C02769=2104.969600,339.035500,-753.612600,90.034588,0.916732,0.000000
C02770=2082.812600,339.026400,-753.612600,88.974616,0.372423,-0.005730
C02771=2027.650200,339.018600,-753.612600,90.756515,-0.183346,-0.000000
C02772=1998.073600,339.007800,-753.612600,89.897078,-0.343775,0.000000
C02773=2074.825300,338.992600,-753.612600,89.358498,1.186023,-0.011459
C02774=2089.149900,338.987500,-753.612600,90.051777,-0.590147,-0.000000
C02775=2053.323900,338.978400,-753.612600,90.332526,-0.332316,-0.000000
C02776=2097.125300,338.974400,-753.612600,90.704949,-0.578687,-0.005730
C02777=2022.267800,338.959500,-753.612600,90.315337,-0.269290,-0.000000
C02778=2024.850700,338.932800,-753.612600,91.318013,0.355234,0.005730
C02779=2085.333300,338.914900,-753.612600,89.891348,0.166158,-0.000000
C02780=2038.206800,338.906800,-753.612600,89.971563,-0.320856,0.000000
C02781=2066.504500,338.886900,-753.612600,90.120532,-0.005730,-0.000000
C02782=2093.534600,338.865200,-753.612600,89.822594,0.091673,-0.000000
C02783=2058.436200,338.801600,-753.612600,90.131991,-0.676090,-0.000000
C02784=2073.063100,338.735200,-803.612600,90.343985,-0.807870,-0.005730
C02785=2062.264800,338.781500,-803.612600,89.364227,0.481285,-0.005730
C02786=2061.218800,338.791200,-803.612600,89.547574,-0.211994,0.000000
C02787=1999.241300,338.815900,-803.612600,88.779810,1.260507,-0.028648
C02788=2061.161000,338.858500,-803.612600,89.203799,0.275020,-0.005730
C02789=2096.996700,338.867600,-803.612600,88.808458,0.372423,-0.005730
C02790=2032.901900,338.882800,-803.612600,89.942915,-0.309397,0.000000
C02791=2104.217500,338.888900,-803.612600,91.174774,1.598552,0.034377
C02792=2019.781000,338.898300,-803.612600,89.587681,0.275020,-0.000000
C02793=2032.219500,338.910500,-803.612600,89.564763,-0.017189,0.000000
C02794=2088.973100,338.917600,-803.612600,90.195016,0.051566,0.000000
C02795=2038.272700,338.924400,-803.612600,89.834053,-0.177617,0.000000
C02796=2014.609200,338.933100,-803.612600,89.862701,-0.252101,0.000000
C02797=2100.091200,338.939200,-803.612600,90.974239,-0.315127,-0.005730
C02798=2046.154000,338.945000,-803.612600,90.842458,-0.807870,-0.011459
C02799=2077.330300,338.949000,-803.612600,89.856971,-0.286479,0.000000
C02800=2071.967600,338.953400,-803.612600,89.742379,0.160428,-0.000000
C02801=1988.870200,338.964600,-803.612600,90.114802,-0.504203,-0.000000
C02802=2111.765200,338.974700,-803.612600,89.983022,0.601606,-0.000000
C02803=2118.654200,338.987200,-803.612600,89.828323,0.068755,-0.000000
C02804=2105.787000,338.990900,-803.612600,90.407010,0.309397,0.000000
C02805=2049.676000,338.996000,-803.612600,90.235123,-0.487014,-0.000000
C02806=2122.801600,339.002700,-803.612600,90.143450,0.521392,0.000000
C02807=1998.518300,339.016900,-803.612600,89.977292,-0.137510,0.000000
C02808=2159.190800,339.028100,-803.612600,90.349715,0.446907,0.000000
C02809=2102.381000,339.034800,-803.612600,90.366903,0.452637,0.005730
C02810=2042.336700,339.040600,-803.612600,89.874160,0.429718,-0.000000
C02811=2113.548000,339.047700,-803.612600,90.143450,0.051566,0.000000
C02812=2131.010900,339.059800,-803.612600,89.484548,0.452637,-0.005730
C02813=1990.465400,339.066600,-803.612600,90.670571,-0.521392,-0.005730
C02814=2154.185700,339.079400,-803.612600,90.492954,0.257831,0.000000
C02815=2103.755700,339.090200,-803.612600,89.879889,0.349504,-0.000000
C02816=1978.876200,339.102600,-803.612600,89.604870,-0.160428,0.000000
C02817=2108.690000,339.109500,-803.612600,89.736650,0.521392,-0.000000
C02818=2117.282000,339.118300,-803.612600,89.157963,0.985487,-0.017189
C02819=2167.864000,339.126700,-803.612600,90.470036,0.469825,0.005730
C02820=1968.699400,339.144300,-803.612600,89.937185,-0.521392,0.000000
C02821=1980.830900,339.149400,-803.612600,89.553303,-0.635983,0.005730
C02822=2012.761200,339.158500,-803.612600,89.312661,-0.234913,0.000000
C02823=1979.519700,339.173400,-803.612600,89.215258,-0.395341,0.005730
C02824=2133.101400,339.181100,-803.612600,90.068965,-0.487014,-0.000000
C02825=2139.307800,339.203900,-803.612600,90.200746,0.721927,0.000000
C02826=2189.894000,339.212200,-803.612600,90.865377,-6.107730,-0.091673
C02827=2164.407500,339.218300,-803.612600,90.779433,-0.131780,-0.000000
C02828=1973.765200,339.226700,-803.612600,88.997534,0.051566,-0.000000
C02829=1963.063900,339.232100,-803.612600,89.793946,-0.120321,0.000000
C02830=2140.823500,339.248700,-803.612600,89.284013,0.693279,-0.011459
C02831=1966.561300,339.257100,-803.612600,90.441388,-0.721927,-0.005730
C02832=2146.546600,339.275400,-803.612600,89.736650,0.469825,-0.000000
C02833=1944.493700,339.305100,-803.612600,89.650706,-0.395341,0.000000
C02834=2164.597400,339.332800,-803.612600,90.934132,0.681820,0.011459
C02835=2179.742100,339.345000,-803.612600,90.630464,1.953786,0.022918
C02836=1959.256700,339.353400,-803.612600,89.845512,-0.315127,0.000000
C02837=1951.206300,339.375000,-803.612600,90.252312,-0.635983,-0.000000
C02838=1940.398000,339.403100,-803.612600,89.839782,-0.590147,0.000000
C02839=1952.858800,339.430500,-803.612600,90.269501,-0.103132,-0.000000
C02840=1940.391000,339.450700,-803.612600,90.172098,-0.676090,-0.000000
C02841=1925.004100,339.506500,-803.612600,90.000210,-0.441178,-0.000000
C02842=1931.783000,339.527400,-803.612600,89.839782,-0.257831,0.000000
C02843=1915.754700,339.565900,-803.612600,89.914267,-0.292208,0.000000
C02844=1925.891500,339.622000,-803.612600,89.541844,-0.538580,0.005730
C02845=1939.013200,339.694600,-803.612600,89.897078,-0.034377,0.000000
C02846=1916.706300,339.756800,-803.612600,90.017399,-0.847978,-0.000000
C02847=1906.137300,339.800400,-803.612600,89.685084,-0.762034,0.005730
C02848=1908.335200,339.879800,-803.612600,89.455901,-0.498473,0.005730
C02849=1891.927500,339.960500,-803.612600,89.748109,-0.985487,0.005730
C02850=1898.280800,340.042000,-803.612600,89.553303,-0.985487,0.005730
C02851=1878.249000,340.138700,-803.612600,90.017399,-1.254778,-0.000000
C02852=1890.381300,340.206100,-803.612600,90.601816,0.406800,0.005730
C02853=1874.073900,340.238200,-803.612600,89.759568,-1.203211,0.005730
C02854=1872.070100,340.338200,-803.612600,89.742379,-0.527121,0.000000
C02855=1878.439100,340.425700,-803.612600,89.983022,-0.842248,0.000000
C02856=1863.563200,340.545000,-803.612600,89.811134,-1.157375,0.005730
C02857=1858.204600,340.602100,-803.612600,90.051777,-1.037054,-0.000000
C02858=1846.137000,340.776800,-803.612600,89.375686,-1.048513,0.011459
C02859=1846.450600,340.848700,-803.612600,89.977292,-1.008406,0.000000
C02860=1839.612500,340.979500,-803.612600,89.146503,-0.355234,0.005730
C02861=1829.812800,341.022700,-803.612600,89.868430,-0.859437,0.000000
C02862=1794.925200,341.065000,-803.612600,91.100289,14.610424,0.280749
C02863=1837.928000,341.117300,-803.612600,89.467360,-0.658901,0.005730
C02864=1824.256700,341.181200,-803.612600,89.564763,-0.676090,0.005730
C02865=1817.402900,341.262300,-803.612600,89.450171,-1.312073,0.011459
C02866=1817.372500,341.325800,-803.612600,90.166368,-1.134456,-0.005730
C02867=1808.346600,341.423100,-803.612600,89.822594,-1.271966,0.005730
C02868=1812.505400,341.463600,-803.612600,89.576222,-1.180293,0.011459
C02869=1798.014800,341.534900,-803.612600,90.217934,5.460288,0.022918
C02870=1798.394100,341.571200,-803.612600,90.452847,4.497719,0.034377
C02871=1798.782000,341.649400,-803.612600,90.733596,3.254400,0.040107
C02872=1798.679300,341.821700,-853.612600,89.089208,2.366316,-0.040107
C02873=1801.796400,341.691700,-853.612600,90.384092,-0.332316,-0.000000
C02874=1803.834000,341.604200,-853.612600,91.358120,-1.976704,-0.045837
C02875=1797.252700,341.515600,-853.612600,93.718707,6.835386,0.441178
C02876=1811.298800,341.443300,-853.612600,90.481495,-1.999623,-0.017189
C02877=1813.044500,341.369400,-853.612600,90.074695,-1.930868,-0.000000
C02878=1814.433300,341.317300,-853.612600,90.510143,-1.673037,-0.017189
C02879=1816.535000,341.199100,-853.612600,90.057506,-0.893814,-0.000000
C02880=1822.945800,341.133500,-853.612600,89.685084,-1.220400,0.005730
C02881=1817.392400,341.111900,-853.612600,90.401281,-1.077161,-0.005730
C02882=1843.858500,340.985200,-853.612600,89.839782,-1.237589,0.005730
C02883=1842.018200,340.879500,-853.612600,90.412740,-1.249048,-0.011459
C02884=1843.463300,340.784900,-853.612600,90.017399,-0.435448,-0.000000
C02885=1850.351600,340.762600,-853.612600,89.954374,-0.888085,0.000000
C02886=1858.825800,340.665300,-853.612600,89.811134,-1.157375,0.005730
C02887=1864.859100,340.596000,-853.612600,89.135044,-0.011459,0.000000
C02888=1864.700800,340.570000,-853.612600,90.292419,-0.796411,-0.005730
C02889=1884.815000,340.449400,-853.612600,89.593410,-0.435448,0.005730
C02890=1866.700100,340.415900,-853.612600,90.945591,-0.733386,-0.011459
C02891=1875.256200,340.323000,-853.612600,90.292419,-0.481285,-0.000000
C02892=1889.321400,340.299700,-853.612600,89.576222,-0.739116,0.005730
C02893=1891.341900,340.243000,-853.612600,89.908537,-1.071431,0.000000
C02894=1897.280800,340.165900,-853.612600,90.848188,-0.635983,-0.011459
C02895=1904.713200,340.119000,-853.612600,89.215258,-0.378152,0.005730
C02896=1934.186200,340.090300,-853.612600,89.404334,-1.094349,0.011459
C02897=1904.887100,340.006800,-853.612600,89.444441,-0.572958,0.005730
C02898=1913.416700,339.981100,-853.612600,89.753839,-0.103132,0.000000
C02899=1924.127800,339.912600,-853.612600,90.607546,-0.045837,-0.000000
C02900=1952.628800,339.828100,-853.612600,87.404712,-0.063025,0.000000
C02901=1953.652400,339.784500,-853.612600,89.650706,-0.389611,0.000000
C02902=1947.297400,339.762600,-853.612600,89.587681,0.063025,-0.000000
C02903=1930.044800,339.732800,-853.612600,89.352768,-0.532851,0.005730
C02904=1937.784000,339.671000,-853.612600,88.819917,-1.014135,0.022918
C02905=1938.403200,339.637200,-853.612600,89.988751,-0.475555,0.000000
C02906=2047.261300,339.589900,-853.612600,77.377950,0.767763,-0.171887
C02907=1962.940900,339.523000,-853.612600,90.023129,-1.008406,-0.000000
C02908=1985.149800,339.488600,-853.612600,88.378740,-0.418259,0.011459
C02909=1981.144300,339.449700,-853.612600,90.023129,-0.613065,-0.000000
C02910=1957.762100,339.410500,-853.612600,89.679354,-0.378152,0.000000
C02911=1990.508900,339.405100,-853.612600,90.131991,-0.171887,-0.000000
C02912=2000.751600,339.354400,-853.612600,89.306932,-0.229183,0.000000
C02913=1982.854200,339.317900,-853.612600,88.739703,-0.492744,0.011459
C02914=2009.978300,339.297300,-853.612600,89.541844,0.767763,-0.005730
C02915=2024.539800,339.284800,-853.612600,90.051777,-0.257831,-0.000000
C02916=2121.511300,339.274700,-853.612600,88.407388,-0.303668,0.005730
C02917=2055.332600,339.230100,-853.612600,90.172098,0.532851,0.000000
C02918=2038.502000,339.213900,-853.612600,89.753839,-0.252101,0.000000
C02919=2083.289400,339.197800,-853.612600,89.352768,0.085944,-0.000000
C02920=1989.215900,339.185900,-853.612600,89.060560,-0.395341,0.005730
C02921=2067.307600,339.179100,-853.612600,89.908537,-0.842248,0.000000
C02922=2188.011000,339.171700,-853.612600,90.624734,-5.036299,-0.057296
C02923=2006.290800,339.150400,-853.612600,88.854295,0.303668,-0.005730
C02924=2087.059600,339.135500,-853.612600,90.939861,-0.842248,-0.011459
C02925=2182.180800,339.129800,-853.612600,89.753839,0.653172,-0.000000
C02926=2165.223600,339.123000,-853.612600,89.736650,0.739116,-0.005730
C02927=2179.411300,339.116900,-853.612600,74.570457,-0.538580,0.148969
C02928=2178.774900,339.105100,-853.612600,91.329473,-0.022918,-0.000000
C02929=1995.124200,339.097000,-853.612600,89.358498,-0.968299,0.011459
C02930=1998.114900,339.089200,-853.612600,90.796622,-0.853707,-0.011459
C02931=2028.129200,339.081800,-853.612600,91.615951,0.332316,0.011459
C02932=2071.745200,339.075700,-853.612600,89.610599,-0.607335,0.005730
C02933=2107.939900,339.069000,-853.612600,90.160639,0.183346,0.000000
C02934=2171.816500,339.059200,-853.612600,89.644977,-0.481285,0.005730
C02935=2006.319000,339.054400,-853.612600,90.716408,-0.441178,-0.005730
C02936=2061.621400,339.046000,-853.612600,89.937185,-0.097403,0.000000
C02937=2092.362100,339.039600,-853.612600,89.650706,-0.687549,0.005730
C02938=2127.230200,339.028800,-853.612600,90.653382,-0.297938,-0.005730
C02939=2142.220100,339.022000,-853.612600,90.080425,0.131780,0.000000
C02940=2050.404100,339.012200,-853.612600,90.366903,-0.097403,-0.000000
C02941=2017.120700,339.008500,-853.612600,91.008616,-0.148969,-0.000000
C02942=2097.055900,339.005400,-853.612600,90.745056,-1.082890,-0.011459
C02943=2146.699300,338.996700,-853.612600,90.195016,-0.378152,-0.000000
C02944=2169.661400,338.991300,-853.612600,90.212205,-0.509932,-0.000000
C02945=2155.902900,338.977700,-853.612600,90.372633,-0.211994,-0.000000
C02946=2135.683800,338.961200,-853.612600,89.862701,0.143239,-0.000000
C02947=2045.946900,338.948700,-853.612600,88.779810,0.819330,-0.017189
C02948=2091.307700,338.939600,-853.612600,89.392875,-0.252101,0.000000
C02949=2072.474700,338.934500,-853.612600,89.994481,-0.956840,0.000000
C02950=2109.023200,338.915600,-853.612600,89.496008,-0.223454,0.000000
C02951=2059.240800,338.906500,-853.612600,89.421523,-0.676090,0.005730
C02952=2189.032800,338.897000,-853.612600,92.091506,-4.251347,-0.154699
C02953=2113.653700,338.883800,-853.612600,90.825270,0.189076,0.000000
C02954=2114.931100,338.865200,-853.612600,85.806159,-0.234913,0.017189
C02955=2141.954900,338.841900,-853.612600,87.324498,-0.137510,0.005730
C02956=2158.166400,338.775700,-853.612600,91.363850,-0.068755,-0.000000
C02957=2182.832600,338.676000,-853.612600,93.770273,-0.269290,-0.017189
C02958=2192.460800,338.381800,-853.612600,92.859270,-14.661990,-0.727656
C02959=1845.943900,-262.579400,-444.761500,-85.135799,-0.796411,179.931666
C02960=2103.620100,-262.360400,-444.761500,-77.847776,0.338045,-179.925936
C02961=2106.924000,-262.167000,-444.761500,-88.086531,0.275020,-179.988962
C02962=1869.037500,-262.039800,-444.761500,-79.022339,1.271966,-179.754049
C02963=2042.284100,-262.001000,-444.761500,-86.321821,1.495420,-179.903018
C02964=2099.976800,-261.979000,-444.761500,-88.579275,1.363640,-179.966043
C02965=2077.569800,-261.892900,-444.761500,-79.474976,-0.378152,179.931666
C02966=2056.224500,-261.862800,-444.761500,-82.248091,-0.555769,179.925936
C02967=1929.876800,-261.815500,-444.761500,-82.654892,1.392287,-179.822804
C02968=1953.938600,-261.752700,-444.761500,-78.403545,-0.784952,179.839993
C02969=2043.564000,-261.713100,-444.761500,-75.722102,-0.802141,179.794156
C02970=1974.190100,-261.625300,-444.761500,-78.667105,-1.673037,179.662376
C02971=1921.842500,-260.819200,-494.761500,-91.965456,0.177617,179.994691
C02972=1911.461000,-260.905300,-494.761500,-92.211828,-0.572958,-179.977503
C02973=1866.999900,-260.969200,-494.761500,-92.165991,-0.613065,-179.977503
C02974=1870.542800,-261.046200,-494.761500,-91.885242,-0.303668,-179.988962
C02975=1916.503500,-261.073900,-494.761500,-91.535737,0.429718,179.988962
C02976=1861.862700,-261.137800,-494.761500,-92.074318,-0.951110,-179.966043
C02977=1937.964400,-261.156000,-494.761500,-91.696166,0.189076,179.994691
C02978=1998.654800,-261.175600,-494.761500,-91.197692,0.206265,179.994691
C02979=2020.094000,-261.188100,-494.761500,-91.535737,-0.423989,-179.988962
C02980=1933.449000,-261.219500,-494.761500,-92.842081,0.154699,179.994691
C02981=2024.472000,-261.238800,-494.761500,-92.343608,-0.120321,-179.994691
C02982=2016.615400,-261.241800,-494.761500,-91.512819,0.263561,179.994691
C02983=1957.998500,-261.260400,-494.761500,-91.742002,0.487014,179.983232
C02984=2090.231400,-261.293500,-494.761500,-91.873782,-0.183346,-179.994691
C02985=1857.870400,-261.303700,-494.761500,-90.899754,0.252101,179.994691
C02986=1869.562400,-261.332000,-494.761500,-91.106019,0.160428,179.994691
C02987=1956.272500,-261.355000,-494.761500,-92.269123,-0.063025,-179.994691
C02988=1980.693200,-261.373900,-494.761500,-91.226340,-0.532851,-179.988962
C02989=2081.434100,-261.394200,-494.761500,-91.060182,-0.022918,-180.000421
C02990=1849.814100,-261.409700,-494.761500,-91.633140,-0.108862,-179.994691
C02991=1898.632500,-261.421900,-494.761500,-91.151856,-0.200535,-179.994691
C02992=2077.098900,-261.431000,-494.761500,-91.128937,-0.647442,-179.988962
C02993=2080.090000,-261.448600,-494.761500,-90.997157,-0.269290,-179.994691
C02994=1868.275200,-261.460100,-494.761500,-91.661788,-0.601606,-179.983232
C02995=1897.656500,-261.478300,-494.761500,-92.498306,2.171510,179.903018
C02996=2006.452600,-261.495900,-494.761500,-91.925349,0.005730,180.000421
C02997=2097.180900,-261.502000,-494.761500,-91.432605,0.275020,179.994691
C02998=2003.950400,-261.515800,-494.761500,-90.378363,0.418259,179.994691
C02999=1974.234800,-261.535800,-494.761500,-90.659112,-0.143239,-180.000421
C03000=2124.803700,-261.548600,-494.761500,-91.656058,0.303668,179.988962
C03001=2094.531400,-261.564500,-494.761500,-90.767974,0.544310,179.994691
C03002=2132.074300,-261.573300,-494.761500,-91.214881,0.338045,179.994691
C03003=1884.756500,-261.584700,-494.761500,-92.647275,-0.567228,-179.971773
C03004=1949.279300,-261.598900,-494.761500,-90.682030,0.498473,179.994691
C03005=1986.413600,-261.603300,-494.761500,-91.329473,0.945380,179.977503
C03006=2088.847000,-261.615200,-494.761500,-90.699219,-0.630254,-179.994691
C03007=1907.677900,-261.626000,-494.761500,-91.323743,-0.217724,-179.994691
C03008=2055.490900,-261.635100,-494.761500,-90.401281,-0.028648,-180.000421
C03009=2026.414700,-261.643900,-494.761500,-90.361174,-0.269290,-180.000421
C03010=2116.655000,-261.651600,-494.761500,-90.504413,0.750575,179.994691
C03011=1933.336100,-261.663800,-494.761500,-91.048723,0.137510,179.994691
C03012=2092.292200,-261.669400,-494.761500,-92.246205,-0.085944,-179.994691
C03013=1945.953800,-261.681700,-494.761500,-91.593033,0.303668,179.988962
C03014=2022.229100,-261.689400,-494.761500,-90.555980,0.492744,179.994691
C03015=2193.443100,-261.697900,-494.761500,-92.630087,-7.563043,-179.656646
C03016=1994.152200,-261.709100,-494.761500,-90.922673,-0.773493,-179.988962
C03017=2117.856500,-261.713800,-494.761500,-90.945591,0.882355,179.983232
C03018=2150.660200,-261.719500,-494.761500,-91.128937,0.126051,180.000421
C03019=2026.671700,-261.724300,-494.761500,-90.212205,0.676090,179.994691
C03020=2181.140100,-261.730400,-494.761500,-89.427253,0.578687,-179.994691
C03021=1954.378200,-261.737500,-494.761500,-90.882565,0.584417,179.988962
C03022=2027.263400,-261.740800,-494.761500,-91.873782,-0.154699,-179.994691
C03023=1902.290500,-261.748100,-494.761500,-91.203422,-0.080214,-180.000421
C03024=2083.758200,-261.758100,-494.761500,-90.332526,-0.498473,-179.994691
C03025=1968.561800,-261.766200,-494.761500,-89.295472,-0.406800,179.994691
C03026=2142.714000,-261.772900,-494.761500,-90.876836,0.452637,179.994691
C03027=2013.614300,-261.780700,-494.761500,-90.836729,-0.796411,-179.988962
C03028=2071.154100,-261.790200,-494.761500,-91.186233,0.275020,179.994691
C03029=2077.380200,-261.803300,-494.761500,-91.644599,0.561499,179.983232
C03030=1914.243800,-261.809100,-494.761500,-90.458577,-0.676090,-179.994691
C03031=2162.444100,-261.814100,-494.761500,-90.916943,0.240642,179.994691
C03032=1989.357100,-261.816500,-494.761500,-90.664842,1.077161,179.988962
C03033=1909.275700,-261.821600,-494.761500,-91.014346,0.074485,180.000421
C03034=2185.796500,-261.830800,-494.761500,-89.954374,0.051566,-180.000421
C03035=1910.961200,-261.834800,-494.761500,-91.415416,-0.103132,-179.994691
C03036=2170.544700,-261.840800,-494.761500,-89.238177,-0.200535,179.994691
C03037=2169.153300,-261.845900,-494.761500,-89.971563,-0.315127,180.000421
C03038=1865.804400,-261.849300,-494.761500,-92.097236,0.647442,179.977503
C03039=1816.495600,-261.851000,-494.761500,-91.850864,-0.899544,-179.971773
C03040=2024.305000,-261.859400,-494.761500,-91.111749,0.229183,179.994691
C03041=2124.318800,-261.865500,-494.761500,-90.934132,0.246372,179.994691
C03042=2080.300500,-261.872100,-494.761500,-90.464306,-0.355234,-179.994691
C03043=2042.447100,-261.881500,-494.761500,-90.229394,-0.326586,-180.000421
C03044=1805.058100,-261.884400,-494.761500,-92.097236,-1.604282,-179.943125
C03045=2172.081100,-261.890800,-494.761500,-90.555980,-0.051566,-180.000421
C03046=2035.399300,-261.894500,-494.761500,-91.071642,0.257831,179.994691
C03047=2175.348700,-261.898300,-494.761500,-90.825270,-0.320856,-179.994691
C03048=2190.438600,-261.904700,-494.761500,-88.986075,-0.951110,179.983232
C03049=2165.547600,-261.916800,-494.761500,-89.983022,-0.853707,180.000421
C03050=2188.317000,-261.922600,-494.761500,-90.452847,0.355234,179.994691
C03051=1810.669700,-261.930200,-494.761500,-91.707625,-1.346451,-179.960314
C03052=2095.544100,-261.934100,-494.761500,-90.762244,-0.870896,-179.988962
C03053=2113.841200,-261.939100,-494.761500,-88.819917,0.315127,-179.994691
C03054=2047.699800,-261.949300,-494.761500,-90.321067,-0.114592,-180.000421
C03055=2038.089400,-261.958100,-494.761500,-89.513196,-0.005730,180.000421
C03056=2022.620600,-261.962800,-494.761500,-90.704949,-0.292208,-179.994691
C03057=2141.279100,-261.973300,-494.761500,-90.177827,0.951110,179.994691
C03058=1879.830200,-261.982700,-494.761500,-91.346661,0.383882,179.988962
C03059=2077.005200,-262.004700,-494.761500,-90.361174,0.028648,180.000421
C03060=1821.697300,-262.022900,-494.761500,-91.180504,-0.687549,-179.983232
C03061=2102.265300,-262.033400,-494.761500,-90.091884,0.091673,180.000421
C03062=1839.440400,-262.042200,-494.761500,-91.638870,0.171887,179.994691
C03063=1920.936600,-262.050300,-494.761500,-84.408142,-0.974028,179.903018
C03064=1848.899200,-262.065200,-494.761500,-89.347039,-1.753251,179.977503
C03065=1811.781100,-262.089400,-494.761500,-91.157585,-1.048513,-179.977503
C03066=1805.613700,-262.106400,-494.761500,-90.767974,-1.283425,-179.983232
C03067=2144.861100,-262.140200,-494.761500,-89.702272,0.166158,-180.000421
C03068=1811.431300,-262.204400,-494.761500,-90.109072,-1.277696,-179.994691
C03069=1863.241200,-262.289800,-494.761500,-90.882565,-0.303668,-179.994691
C03070=1831.979100,-262.356000,-494.761500,-93.277529,0.504203,179.971773
C03071=1796.446100,-262.384400,-494.761500,-90.578898,5.826981,179.943125
C03072=1847.265200,-262.436800,-494.761500,-91.060182,-1.100079,-179.977503
C03073=1818.793200,-262.555400,-494.761500,-91.489901,-0.796411,-179.977503
C03074=1801.917400,-262.590200,-494.761500,-91.862323,-1.340721,-179.954584
C03075=1806.287400,-262.817200,-494.761500,-77.418057,-2.326209,179.479029
C03076=2193.404700,-262.778700,-544.761500,-88.166746,1.770440,-179.943125
C03077=2189.447400,-261.928300,-544.761500,-90.813811,4.360209,179.937396
C03078=2190.414600,-261.848900,-544.761500,-90.619005,0.418259,179.994691
C03079=2184.051200,-261.800300,-544.761500,-89.960103,-1.048513,180.000421
C03080=2181.482000,-261.731400,-544.761500,-90.693489,0.699009,179.988962
C03081=2167.358100,-261.706900,-544.761500,-90.699219,-0.120321,-180.000421
C03082=2171.713400,-261.665800,-544.761500,-90.762244,0.126051,180.000421
C03083=2156.638400,-261.640200,-544.761500,-91.002887,0.744845,179.988962
C03084=2139.836100,-261.607700,-544.761500,-91.289365,0.137510,179.994691
C03085=1812.547300,-261.579000,-544.761500,-91.237799,-1.741792,-179.960314
C03086=2171.946200,-261.543500,-544.761500,-90.859647,1.231859,179.983232
C03087=2154.229600,-261.503000,-544.761500,-91.077371,0.699009,179.988962
C03088=2173.622000,-261.451600,-544.761500,-91.318013,0.693279,179.983232
C03089=1814.094900,-261.418500,-544.761500,-90.716408,-1.082890,-179.988962
C03090=1805.093300,-261.396200,-544.761500,-91.065912,-1.398017,-179.971773
C03091=2168.330700,-261.378000,-544.761500,-90.985698,1.025594,179.983232
C03092=1836.531800,-261.352000,-544.761500,-91.713354,-0.624524,-179.983232
C03093=2178.750100,-261.297200,-544.761500,-90.498684,1.741792,179.983232
C03094=2100.472100,-261.271900,-544.761500,-91.512819,0.263561,179.994691
C03095=2129.860700,-261.209700,-544.761500,-92.206098,0.355234,179.988962
C03096=1809.421600,-261.193900,-544.761500,-90.492954,-0.933921,-179.994691
C03097=2164.807600,-261.175600,-544.761500,-90.309608,1.306344,179.994691
C03098=1821.197500,-261.137100,-544.761500,-90.739326,-0.916732,-179.988962
C03099=2064.002700,-261.115500,-544.761500,-91.495630,-0.085944,-180.000421
C03100=1837.038600,-261.079700,-544.761500,-91.289365,-0.796411,-179.983232
C03101=2144.955900,-261.059100,-544.761500,-91.587304,0.670361,179.983232
C03102=1816.312600,-261.036800,-544.761500,-90.573168,-0.681820,-179.994691
C03103=2007.052200,-261.008700,-544.761500,-91.232070,1.289155,179.971773
C03104=1815.077400,-260.995200,-544.761500,-91.106019,-1.254778,-179.977503
C03105=2020.728300,-260.981300,-544.761500,-91.684706,0.401070,179.988962
C03106=1935.614200,-260.958400,-544.761500,-91.827946,0.395341,179.988962
C03107=1815.197000,-260.941800,-544.761500,-89.581951,-1.988164,179.983232
C03108=2038.539300,-260.917200,-544.761500,-92.377985,0.584417,179.977503
C03109=1995.584900,-260.905300,-544.761500,-92.693112,0.315127,179.983232
C03110=1821.920700,-260.891500,-544.761500,-91.111749,-1.157375,-179.977503
C03111=1972.452200,-260.872900,-544.761500,-91.661788,0.183346,179.994691
C03112=1871.622600,-260.855000,-544.761500,-91.839405,-0.223454,-179.994691
C03113=1992.617400,-260.839600,-544.761500,-93.162937,0.074485,179.994691
C03114=2131.634500,-260.824600,-544.761500,-91.656058,0.779223,179.977503
C03115=2035.438300,-260.806300,-544.761500,-91.037264,-0.933921,-179.983232
C03116=2114.512500,-260.763800,-544.761500,-91.421146,1.128727,179.971773
C03117=2078.864700,-260.750300,-544.761500,-92.171721,0.297938,179.988962
C03118=2157.676000,-260.733700,-544.761500,-91.318013,1.707414,179.960314
C03119=1866.480200,-260.724600,-544.761500,-91.226340,-0.647442,-179.988962
C03120=1988.083400,-260.707700,-544.761500,-91.805028,0.246372,179.994691
C03121=1978.238600,-260.688100,-544.761500,-91.673247,0.739116,179.977503
C03122=1897.058900,-260.662000,-544.761500,-92.859270,-1.306344,-179.937396
C03123=1825.113400,-260.652600,-544.761500,-90.876836,-0.951110,-179.983232
C03124=2095.767400,-260.644900,-544.761500,-91.633140,0.544310,179.983232
C03125=1876.881500,-260.633000,-544.761500,-92.836352,0.739116,179.966043
C03126=2074.786700,-260.610100,-544.761500,-92.194639,0.561499,179.977503
C03127=1924.829500,-260.589100,-544.761500,-91.186233,-0.389611,-179.994691
C03128=2116.875600,-260.582700,-544.761500,-91.976915,0.143239,179.994691
C03129=1842.483900,-260.561400,-544.761500,-91.163315,-1.243318,-179.977503
C03130=2027.544200,-260.536400,-544.761500,-91.873782,0.343775,179.988962
C03131=1850.823900,-260.517500,-544.761500,-91.243529,-0.068755,-180.000421
C03132=1875.209900,-260.495900,-544.761500,-91.902430,-0.177617,-179.994691
C03133=1971.870300,-260.470500,-544.761500,-91.363850,0.338045,179.994691
C03134=1987.957000,-260.444900,-544.761500,-91.174774,2.234535,179.954584
C03135=1835.514400,-260.423200,-544.761500,-89.919996,-0.968299,180.000421
C03136=1980.580000,-260.409000,-544.761500,-92.504036,-0.739116,-179.966043
C03137=1848.362100,-260.392500,-544.761500,-91.484171,-0.802141,-179.977503
C03138=1831.829900,-260.365800,-544.761500,-89.730920,-2.881978,179.988962
C03139=2135.648000,-260.354300,-544.761500,-91.403957,0.584417,179.983232
C03140=1920.149600,-260.334400,-544.761500,-92.137343,0.252101,179.988962
C03141=1873.512100,-260.317800,-544.761500,-91.083101,-0.515662,-179.988962
C03142=2090.011200,-260.305000,-544.761500,-92.097236,0.257831,179.988962
C03143=1999.619000,-260.288600,-544.761500,-91.501360,-0.097403,-179.994691
C03144=2118.771400,-260.267500,-544.761500,-91.232070,0.790682,179.983232
C03145=1893.437100,-260.253300,-544.761500,-91.598763,-0.303668,-179.988962
C03146=1995.325000,-260.237900,-544.761500,-92.635816,-0.206265,-179.988962
C03147=1877.827800,-260.217500,-544.761500,-91.363850,-1.111538,-179.971773
C03148=1861.590800,-260.198900,-544.761500,-92.114425,-0.561499,-179.977503
C03149=1949.022700,-260.188100,-544.761500,-91.931078,0.045837,180.000421
C03150=2065.874400,-260.160700,-544.761500,-92.188909,0.223454,179.988962
C03151=1984.529000,-260.117400,-544.761500,-91.638870,-0.418259,-179.988962
C03152=1946.014500,-260.067500,-544.761500,-91.919619,-0.085944,-179.994691
C03153=2028.490500,-260.046200,-544.761500,-90.945591,1.461042,179.977503
C03154=1878.387900,-260.014800,-544.761500,-91.495630,-1.134456,-179.971773
C03155=2054.593000,-260.005000,-544.761500,-92.750408,-0.332316,-179.983232
C03156=2072.406500,-259.984400,-544.761500,-92.429552,-0.022918,-180.000421
C03157=1954.819400,-259.971500,-544.761500,-92.767597,-0.349504,-179.983232
C03158=2079.669100,-259.920900,-544.761500,-92.148802,0.120321,179.994691
C03159=2034.819700,-259.900600,-544.761500,-92.830622,0.326586,179.983232
C03160=2001.013700,-259.884400,-544.761500,-90.727867,0.504203,179.994691
C03161=1936.039800,-259.870200,-544.761500,-92.412363,-0.389611,-179.983232
C03162=2016.505000,-259.830600,-544.761500,-91.461253,-1.329262,-179.966043
C03163=2105.713500,-259.797200,-544.761500,-92.292042,0.681820,179.971773
C03164=1928.160200,-259.790800,-544.761500,-92.337878,0.521392,179.977503
C03165=2100.667200,-259.760700,-544.761500,-92.589980,0.338045,179.983232
C03166=1968.585700,-259.715800,-544.761500,-92.549873,1.919409,179.914477
C03167=1957.890100,-259.692800,-544.761500,-92.446740,1.111538,179.954584
C03168=1907.944600,-259.650900,-544.761500,-92.412363,-0.928192,-179.960314
C03169=2022.531700,-259.635000,-544.761500,-91.644599,-0.269290,-179.994691
C03170=2045.046000,-259.595200,-544.761500,-91.879512,-0.882355,-179.971773
C03171=1945.854800,-259.558700,-544.761500,-93.816109,0.618794,179.960314
C03172=2035.480500,-259.537400,-544.761500,-92.229016,0.807870,179.966043
C03173=2051.644000,-259.510700,-544.761500,-92.504036,-0.784952,-179.966043
C03174=2087.205400,-259.470800,-544.761500,-91.232070,0.349504,179.994691
C03175=1976.162800,-259.450000,-544.761500,-93.374932,0.481285,179.971773
C03176=1946.439700,-259.404300,-544.761500,-91.673247,-0.114592,-179.994691
C03177=1957.313100,-259.374000,-544.761500,-92.028481,-0.498473,-179.983232
C03178=2083.156000,-259.348500,-544.761500,-90.762244,-0.040107,-180.000421
C03179=1979.022000,-259.233300,-544.761500,-90.722137,-0.120321,-180.000421
C03180=1975.506000,-257.856600,-594.761500,-92.108695,-0.389611,-179.983232
C03181=2006.601900,-257.960700,-594.761500,-91.552926,0.819330,179.977503
C03182=2043.583500,-257.974500,-594.761500,-90.796622,0.000000,180.000421
C03183=2076.505700,-257.997800,-594.761500,-91.191963,0.572958,179.988962
C03184=2005.853900,-258.029900,-594.761500,-91.999833,0.177617,179.994691
C03185=1968.632200,-258.047200,-594.761500,-91.020075,0.148969,179.994691
C03186=1950.789900,-258.061700,-594.761500,-91.650329,-0.171887,-179.994691
C03187=1936.259000,-258.086700,-594.761500,-91.117478,0.699009,179.988962
C03188=1945.613800,-258.125400,-594.761500,-91.959726,-1.804817,-179.937396
C03189=2075.447500,-258.155600,-594.761500,-91.123208,-0.080214,-180.000421
C03190=1950.546200,-258.173200,-594.761500,-92.383715,-0.664631,-179.971773
C03191=1926.315400,-258.193800,-594.761500,-90.767974,-0.383882,-179.994691
C03192=1982.653400,-258.200200,-594.761500,-90.596087,0.739116,179.994691
C03193=1978.382700,-258.235700,-594.761500,-91.959726,-0.103132,-179.994691
C03194=2019.060400,-258.261000,-594.761500,-91.547197,-0.103132,-179.994691
C03195=1947.702100,-258.288000,-594.761500,-91.295095,-0.034377,-180.000421
C03196=2010.528200,-258.308000,-594.761500,-90.636194,-0.590147,-179.994691
C03197=1974.208100,-258.315100,-594.761500,-91.386768,-0.246372,-179.994691
C03198=2047.057400,-258.336700,-594.761500,-90.756515,0.710468,179.988962
C03199=2110.855600,-258.380300,-594.761500,-90.533061,1.363640,179.988962
C03200=1897.268300,-258.412700,-594.761500,-91.077371,0.847978,179.983232
C03201=1934.923000,-258.446500,-594.761500,-90.928402,-0.211994,-179.994691
C03202=2062.708900,-258.475500,-594.761500,-92.876459,-1.008406,-179.948855
C03203=1991.921800,-258.489100,-594.761500,-90.991427,-0.040107,-180.000421
C03204=2071.862000,-258.515800,-594.761500,-91.438335,0.057296,180.000421
C03205=2077.376000,-258.534000,-594.761500,-92.068588,0.859437,179.971773
C03206=1885.348400,-258.538000,-594.761500,-89.702272,0.131780,-180.000421
C03207=1982.583000,-258.548200,-594.761500,-91.478442,-0.584417,-179.983232
C03208=1900.176200,-258.564700,-594.761500,-91.289365,-0.068755,-180.000421
C03209=1966.706900,-258.589400,-594.761500,-90.813811,0.762034,179.988962
C03210=2107.198600,-258.596500,-594.761500,-90.997157,0.458366,179.994691
C03211=2059.464300,-258.620500,-594.761500,-91.340932,-0.103132,-180.000421
C03212=1910.029600,-258.641800,-594.761500,-91.432605,-0.446907,-179.988962
C03213=2118.898600,-258.685700,-594.761500,-90.853918,1.289155,179.983232
C03214=1883.168600,-258.709000,-594.761500,-91.060182,-0.756304,-179.983232
C03215=2032.730800,-258.733300,-594.761500,-91.890971,0.338045,179.988962
C03216=2039.315900,-258.747200,-594.761500,-92.217557,0.011459,180.000421
C03217=1906.954400,-258.789700,-594.761500,-92.314960,0.189076,179.994691
C03218=2122.856000,-258.799900,-594.761500,-90.332526,1.569904,179.988962
C03219=1937.499100,-258.819800,-594.761500,-91.742002,0.429718,179.988962
C03220=2076.275000,-258.844800,-594.761500,-91.799298,0.607335,179.983232
C03221=2006.823400,-258.871500,-594.761500,-90.876836,0.223454,179.994691
C03222=1892.551100,-258.879900,-594.761500,-91.398227,-0.687549,-179.983232
C03223=2014.743300,-258.919500,-594.761500,-91.369580,0.584417,179.983232
C03224=2074.409200,-258.971800,-594.761500,-92.521225,0.355234,179.983232
C03225=1921.246800,-258.981000,-594.761500,-91.495630,0.045837,180.000421
C03226=2056.623300,-259.012400,-594.761500,-92.309230,0.790682,179.966043
C03227=1976.930800,-259.023200,-594.761500,-91.060182,-0.326586,-179.994691
C03228=1888.774200,-259.039100,-594.761500,-91.197692,-1.002676,-179.977503
C03229=1875.304000,-259.056300,-594.761500,-91.707625,-0.223454,-179.994691
C03230=1907.160300,-259.075600,-594.761500,-92.286312,0.017189,180.000421
C03231=1887.079600,-259.105600,-594.761500,-90.762244,-1.243318,-179.983232
C03232=1936.288600,-259.118800,-594.761500,-92.435281,0.383882,179.983232
C03233=2040.977100,-259.134300,-594.761500,-90.945591,-0.343775,-179.994691
C03234=2128.164300,-259.163700,-594.761500,-91.398227,1.300614,179.966043
C03235=2072.801000,-259.188400,-594.761500,-92.137343,0.429718,179.983232
C03236=1871.532200,-259.218100,-594.761500,-90.767974,-1.988164,-179.971773
C03237=2034.112800,-259.246800,-594.761500,-91.994104,-0.131780,-179.994691
C03238=1862.458300,-259.269800,-594.761500,-91.587304,-1.403747,-179.960314
C03239=1857.782200,-259.295500,-594.761500,-91.048723,-1.764710,-179.966043
C03240=1964.076700,-259.322500,-594.761500,-92.102966,0.767763,179.971773
C03241=2047.145300,-259.352600,-594.761500,-92.853540,-1.386558,-179.931666
C03242=1880.959500,-259.406300,-594.761500,-91.426875,-0.796411,-179.977503
C03243=2004.925400,-259.456300,-594.761500,-91.598763,0.928192,179.971773
C03244=2099.609400,-259.488400,-594.761500,-91.776380,2.051189,179.937396
C03245=2144.537300,-259.524200,-594.761500,-90.842458,2.354857,179.966043
C03246=2105.933800,-259.586700,-594.761500,-92.039940,0.595876,179.977503
C03247=1848.169700,-259.648900,-594.761500,-90.074695,-1.873572,-180.000421
C03248=1847.758100,-259.734400,-594.761500,-90.550250,-1.610011,-179.983232
C03249=2144.235100,-259.767100,-594.761500,-91.518549,2.515285,179.931666
C03250=1842.596100,-259.859400,-594.761500,-90.796622,-1.375099,-179.983232
C03251=2136.079200,-259.888100,-594.761500,-91.530008,1.575634,179.960314
C03252=2143.069900,-259.985700,-594.761500,-91.581574,1.541256,179.960314
C03253=1840.442500,-260.007300,-594.761500,-90.074695,-2.343397,-179.994691
C03254=1836.528600,-260.061400,-594.761500,-90.389822,-2.011082,-179.988962
C03255=2161.067000,-260.162800,-594.761500,-89.948644,3.277319,-179.994691
C03256=1833.421400,-260.234000,-594.761500,-90.349715,-2.761657,-179.983232
C03257=2156.691400,-260.301300,-594.761500,-91.318013,1.919409,179.954584
C03258=1828.131500,-260.435400,-594.761500,-90.487225,0.343775,179.994691
C03259=1822.949300,-260.521200,-594.761500,-90.401281,-2.320479,-179.983232
C03260=2169.354800,-260.567500,-594.761500,-90.000210,2.945003,180.000421
C03261=1820.066800,-260.698600,-594.761500,-89.771027,-1.873572,179.994691
C03262=1821.878900,-260.763800,-594.761500,-90.154909,-2.452259,-179.994691
C03263=1815.778300,-260.860400,-594.761500,-89.295472,-1.913679,179.977503
C03264=2176.814800,-260.934000,-594.761500,-90.676301,3.254400,179.960314
C03265=2172.570400,-260.978500,-594.761500,-90.567439,2.274642,179.977503
C03266=1809.014800,-261.035700,-594.761500,-90.005940,-2.062648,-180.000421
C03267=1812.378300,-261.091800,-594.761500,-89.994481,-2.486637,180.000421
C03268=1811.469600,-261.134100,-594.761500,-89.587681,-3.030947,179.977503
C03269=1806.242800,-261.193900,-594.761500,-89.129315,-2.354857,179.966043
C03270=1799.144000,-261.309100,-594.761500,-88.991805,-3.288778,179.943125
C03271=1796.063900,-261.353000,-594.761500,-88.126638,7.465640,-179.754049
C03272=1800.022000,-261.367200,-594.761500,-88.900131,-1.764710,179.966043
C03273=1802.737100,-261.531700,-594.761500,-89.381416,-3.065324,179.966043
C03274=1795.613900,-261.580000,-594.761500,-87.215636,0.653172,-179.966043
C03275=2187.688400,-261.652000,-594.761500,-89.856971,3.432017,-179.988962
C03276=1797.468200,-261.768900,-594.761500,-88.877213,-2.876248,179.943125
C03277=2190.839400,-261.875000,-594.761500,-91.031534,1.535527,179.971773
C03278=1797.016500,-261.995900,-594.761500,-88.860024,2.893437,-179.943125
C03279=1798.970800,-262.465800,-644.761500,-88.814188,-2.692902,179.943125
C03280=1796.247600,-262.211100,-644.761500,-89.547574,-0.401070,179.994691
C03281=2191.211700,-262.002300,-644.761500,-87.536492,-0.080214,179.994691
C03282=1803.707200,-261.891800,-644.761500,-89.679354,-5.993139,179.966043
C03283=1803.478200,-261.793900,-644.761500,-89.398605,-3.277319,179.966043
C03284=2187.072000,-261.722600,-644.761500,-88.825647,4.182592,-179.914477
C03285=2193.651900,-261.661800,-644.761500,-91.976915,-13.676503,-179.530596
C03286=2187.221700,-261.583900,-644.761500,-89.713732,3.460665,-179.983232
C03287=1804.257500,-261.440800,-644.761500,-90.544520,-4.572203,-179.954584
C03288=1811.483600,-261.369500,-644.761500,-89.077748,-3.982057,179.937396
C03289=1810.682200,-261.260800,-644.761500,-90.779433,-2.933544,-179.960314
C03290=2177.467100,-261.107200,-644.761500,-90.154909,3.827358,179.988962
C03291=2177.509300,-260.994500,-644.761500,-89.702272,3.179916,-179.983232
C03292=1821.215600,-260.865200,-644.761500,-90.097613,-2.927814,-179.994691
C03293=2172.041700,-260.749300,-644.761500,-89.742379,3.105431,-179.988962
C03294=2170.868000,-260.702800,-644.761500,-90.286689,3.093972,179.983232
C03295=1828.065600,-260.492800,-644.761500,-91.163315,-3.008028,-179.937396
C03296=1832.099000,-260.313800,-644.761500,-90.424199,-3.225752,-179.977503
C03297=2164.047100,-260.166500,-644.761500,-88.751162,2.796034,-179.937396
C03298=1836.783100,-260.034700,-644.761500,-89.627788,-2.589769,179.983232
C03299=2156.915300,-259.932300,-644.761500,-89.759568,2.635606,-179.988962
C03300=1842.827200,-259.797500,-644.761500,-90.149179,-3.168457,-179.988962
C03301=1836.341800,-259.756700,-644.761500,-91.323743,-1.776169,-179.960314
C03302=1845.845400,-259.557700,-644.761500,-89.392875,-3.970598,179.960314
C03303=1850.073800,-259.457700,-644.761500,-90.286689,-2.641335,-179.988962
C03304=1853.851300,-259.396200,-644.761500,-90.624734,-1.942327,-179.977503
C03305=1847.099300,-259.295200,-644.761500,-89.077748,-2.870519,179.954584
C03306=2141.896000,-259.242500,-644.761500,-89.673625,2.824682,-179.983232
C03307=1856.964600,-259.117800,-644.761500,-90.275230,-2.217347,-179.988962
C03308=1861.627400,-259.005600,-644.761500,-89.243906,-2.595499,179.966043
C03309=1859.827900,-258.931000,-644.761500,-90.510143,-2.171510,-179.983232
C03310=1871.831800,-258.822500,-644.761500,-90.057506,-1.764710,-180.000421
C03311=1865.678800,-258.764100,-644.761500,-89.427253,-1.598552,179.983232
C03312=2122.715500,-258.728600,-644.761500,-91.008616,1.363640,179.977503
C03313=2117.886100,-258.659000,-644.761500,-89.524655,2.034000,-179.983232
C03314=1871.010900,-258.626900,-644.761500,-90.292419,-2.383504,-179.988962
C03315=1876.193500,-258.563000,-644.761500,-91.421146,-1.718873,-179.954584
C03316=2116.714400,-258.509800,-644.761500,-91.209151,0.641713,179.988962
C03317=1885.146900,-258.430600,-644.761500,-91.988374,-1.885031,-179.937396
C03318=2114.671400,-258.362400,-644.761500,-90.189287,1.386558,179.994691
C03319=1872.610800,-258.298500,-644.761500,-90.848188,-1.701685,-179.977503
C03320=1882.136000,-258.248200,-644.761500,-89.559033,-1.822006,179.983232
C03321=1895.852800,-258.212700,-644.761500,-90.166368,-1.443854,-179.994691
C03322=1889.422500,-258.161400,-644.761500,-90.916943,-1.065701,-179.983232
C03323=2102.364000,-258.132500,-644.761500,-89.839782,0.773493,-180.000421
C03324=2101.942600,-258.108000,-644.761500,-90.126261,0.899544,180.000421
C03325=1899.936700,-258.068100,-644.761500,-90.407010,-1.082890,-179.994691
C03326=2103.695400,-258.025200,-644.761500,-89.788216,1.140186,-179.994691
C03327=2082.194000,-257.993100,-644.761500,-91.209151,1.443854,179.971773
C03328=2076.015400,-257.952900,-644.761500,-90.515872,0.727656,179.994691
C03329=1910.703300,-257.931300,-644.761500,-91.060182,-0.452637,-179.988962
C03330=1917.100900,-257.917700,-644.761500,-90.785163,-0.389611,-179.994691
C03331=1940.719100,-257.905200,-644.761500,-91.306554,-0.269290,-179.994691
C03332=1961.928100,-257.889700,-644.761500,-91.146126,0.263561,179.994691
C03333=2090.408800,-257.871800,-644.761500,-90.584627,0.939651,179.988962
C03334=2072.946000,-257.854600,-644.761500,-90.384092,1.340721,179.988962
C03335=1910.699500,-257.840400,-644.761500,-88.923050,0.905273,-179.983232
C03336=2023.164200,-257.823500,-644.761500,-91.002887,-0.017189,-180.000421
C03337=2084.155600,-257.804900,-644.761500,-90.813811,0.343775,179.994691
C03338=2012.223800,-257.788000,-644.761500,-91.593033,-0.034377,-180.000421
C03339=1936.512200,-257.780800,-644.761500,-90.670571,-0.223454,-179.994691
C03340=1919.876700,-257.759300,-644.761500,-90.750785,-0.853707,-179.988962
C03341=2002.111600,-257.748500,-644.761500,-90.246582,-0.664631,-179.994691
C03342=2018.400300,-257.732300,-644.761500,-91.123208,0.515662,179.988962
C03343=2064.837500,-257.722200,-644.761500,-89.793946,0.550039,-180.000421
C03344=2081.925200,-257.710300,-644.761500,-89.518926,0.366693,-179.994691
C03345=2037.211000,-257.700900,-644.761500,-90.429929,-0.916732,-179.994691
C03346=1993.727300,-257.689700,-644.761500,-91.426875,-0.103132,-179.994691
C03347=2001.922300,-257.685300,-644.761500,-90.997157,0.412530,179.994691
C03348=1930.788900,-257.678600,-644.761500,-91.289365,-0.521392,-179.988962
C03349=1900.989700,-257.669100,-644.761500,-91.449794,-0.796411,-179.977503
C03350=1937.710700,-257.660000,-644.761500,-90.682030,-0.418259,-179.994691
C03351=2083.356000,-257.652200,-644.761500,-90.252312,0.418259,180.000421
C03352=1967.410700,-257.646100,-644.761500,-91.169044,-0.297938,-179.994691
C03353=1925.347400,-257.641100,-644.761500,-90.538791,-0.825059,-179.994691
C03354=1958.648200,-257.624900,-644.761500,-91.008616,0.240642,179.994691
C03355=2037.434100,-257.617800,-644.761500,-91.254988,-0.080214,-180.000421
C03356=1899.387800,-257.605600,-644.761500,-90.504413,-1.346451,-179.988962
C03357=2025.422700,-257.589700,-644.761500,-92.011292,0.527121,179.983232
C03358=1975.027400,-257.575900,-644.761500,-91.913889,1.822006,179.937396
C03359=1915.038200,-257.549200,-644.761500,-90.349715,-0.676090,-179.994691
C03360=1972.643600,-257.539400,-644.761500,-91.031534,0.750575,179.988962
C03361=1959.202700,-257.523500,-644.761500,-91.031534,1.220400,179.977503
C03362=1951.110200,-257.510000,-644.761500,-90.212205,-0.011459,-180.000421
C03363=2010.252000,-257.502200,-644.761500,-89.392875,-0.515662,179.994691
C03364=1928.495500,-257.494400,-644.761500,-91.088830,0.378152,179.994691
C03365=2029.678300,-257.485000,-644.761500,-91.094560,-0.452637,-179.988962
C03366=1953.653200,-257.474800,-644.761500,-90.057506,-0.320856,-180.000421
C03367=1941.790800,-257.458300,-644.761500,-90.412740,-0.017189,-180.000421
C03368=2020.357300,-257.444100,-644.761500,-90.246582,0.389611,180.000421
C03369=2043.800600,-257.430600,-644.761500,-89.547574,-1.122997,179.988962
C03370=1953.336000,-257.408000,-644.761500,-91.037264,0.080214,180.000421
C03371=1974.292200,-257.387300,-644.761500,-89.965833,0.120321,-180.000421
C03372=1965.413900,-257.369800,-644.761500,-90.470036,-1.025594,-179.988962
C03373=2005.907100,-257.337000,-644.761500,-91.295095,-0.555769,-179.988962
C03374=1967.602900,-257.314700,-644.761500,-90.200746,-0.103132,-180.000421
C03375=1947.102600,-257.138400,-694.761500,-90.871106,0.332316,179.994691
C03376=1999.192800,-257.207300,-694.761500,-90.475765,0.320856,179.994691
C03377=1948.866600,-257.230900,-694.761500,-89.266824,0.080214,-180.000421
C03378=1942.446700,-257.262000,-694.761500,-89.828323,-0.303668,180.000421
C03379=1955.709400,-257.274300,-694.761500,-89.748109,0.343775,-180.000421
C03380=2008.496600,-257.286700,-694.761500,-90.149179,-0.063025,-180.000421
C03381=1985.093300,-257.298500,-694.761500,-89.771027,-0.034377,180.000421
C03382=1921.908300,-257.314700,-694.761500,-89.748109,0.171887,-180.000421
C03383=1933.695100,-257.326500,-694.761500,-89.673625,-0.647442,179.994691
C03384=1928.511500,-257.341400,-694.761500,-89.713732,-0.131780,180.000421
C03385=2015.374900,-257.357300,-694.761500,-89.742379,-0.034377,180.000421
C03386=1972.311300,-257.364000,-694.761500,-89.879889,0.022918,-180.000421
C03387=2013.357200,-257.370800,-694.761500,-90.407010,0.154699,180.000421
C03388=1942.638100,-257.379900,-694.761500,-89.238177,0.108862,-180.000421
C03389=2030.388300,-257.394100,-694.761500,-89.369957,0.211994,-180.000421
C03390=2023.263300,-257.401200,-694.761500,-88.544898,0.206265,-179.994691
C03391=1993.455900,-257.407300,-694.761500,-90.258041,0.349504,180.000421
C03392=1914.113500,-257.412700,-694.761500,-89.811134,-0.739116,179.994691
C03393=1957.645800,-257.418400,-694.761500,-88.636571,0.028648,-180.000421
C03394=1915.229900,-257.423800,-694.761500,-89.679354,-0.332316,180.000421
C03395=2035.118000,-257.430300,-694.761500,-90.160639,1.306344,179.994691
C03396=2042.432900,-257.437700,-694.761500,-89.788216,-1.134456,179.994691
C03397=1960.369600,-257.459600,-694.761500,-89.788216,0.355234,-180.000421
C03398=1912.767400,-257.480600,-694.761500,-90.412740,-0.160428,-180.000421
C03399=1920.555300,-257.490400,-694.761500,-90.240853,-0.068755,-180.000421
C03400=2049.461400,-257.496500,-694.761500,-89.518926,0.790682,-179.994691
C03401=1909.195800,-257.516400,-694.761500,-89.811134,-0.206265,180.000421
C03402=2035.464800,-257.533600,-694.761500,-89.599140,0.435448,-179.994691
C03403=1905.283100,-257.545800,-694.761500,-90.767974,-0.756304,-179.988962
C03404=2030.623500,-257.556600,-694.761500,-88.980346,-0.544310,179.988962
C03405=1890.242300,-257.577900,-694.761500,-90.349715,-0.922462,-179.994691
C03406=2025.437200,-257.603600,-694.761500,-88.940239,1.100079,-179.977503
C03407=2041.125200,-257.627200,-694.761500,-89.679354,-1.398017,179.994691
C03408=1984.875400,-257.644400,-694.761500,-89.003264,0.234913,-179.994691
C03409=1898.180100,-257.657300,-694.761500,-90.338256,0.017189,180.000421
C03410=2066.220800,-257.669100,-694.761500,-89.679354,0.257831,-180.000421
C03411=2074.116800,-257.694400,-694.761500,-89.759568,0.590147,-179.994691
C03412=1888.206100,-257.725500,-694.761500,-90.957050,-1.690225,-179.971773
C03413=2062.616200,-257.755300,-694.761500,-89.289743,0.166158,-180.000421
C03414=2045.907200,-257.785300,-694.761500,-89.272554,0.555769,-179.994691
C03415=1889.336400,-257.813700,-694.761500,-90.051777,-1.673037,-180.000421
C03416=2031.982900,-257.833000,-694.761500,-89.358498,-0.229183,179.994691
C03417=2052.273100,-257.864000,-694.761500,-88.945968,0.945380,-179.983232
C03418=2083.032200,-257.899500,-694.761500,-89.100667,1.134456,-179.983232
C03419=2092.348800,-257.944500,-694.761500,-89.261095,1.329262,-179.983232
C03420=1884.475600,-257.982000,-694.761500,-91.421146,-1.266237,-179.966043
C03421=1869.344500,-258.030600,-694.761500,-90.240853,-1.713144,-179.994691
C03422=1868.652000,-258.054600,-694.761500,-92.074318,-0.063025,-180.000421
C03423=2058.761600,-258.080900,-694.761500,-88.837106,1.283425,-179.971773
C03424=1862.957400,-258.152200,-694.761500,-90.000210,-1.398017,180.000421
C03425=2090.167300,-258.202600,-694.761500,-88.751162,0.905273,-179.977503
C03426=2069.807400,-258.251000,-694.761500,-88.751162,0.452637,-179.988962
C03427=1870.433100,-258.324500,-694.761500,-90.619005,-1.071431,-179.988962
C03428=2089.421100,-258.392100,-694.761500,-88.711055,0.830789,-179.983232
C03429=2096.217000,-258.445100,-694.761500,-89.060560,1.398017,-179.977503
C03430=1850.421700,-258.527200,-694.761500,-90.063236,-2.119944,-180.000421
C03431=1851.975500,-258.646500,-694.761500,-90.859647,-2.652795,-179.960314
C03432=2120.879400,-258.712400,-694.761500,-89.748109,-0.068755,180.000421
C03433=1846.345100,-258.807000,-694.761500,-90.298149,-1.896490,-179.988962
C03434=1843.146100,-258.826900,-694.761500,-90.750785,-2.079837,-179.971773
C03435=1845.750800,-258.936700,-694.761500,-91.025805,-2.240265,-179.960314
C03436=2128.259800,-259.010000,-694.761500,-89.685084,1.919409,-179.988962
C03437=1833.874500,-259.039800,-694.761500,-90.985698,-2.841871,-179.948855
C03438=2133.807600,-259.216800,-694.761500,-89.289743,1.970975,-179.977503
C03439=1838.098800,-259.285400,-694.761500,-90.876836,-2.360586,-179.966043
C03440=2117.638300,-259.365800,-694.761500,-88.636571,1.632930,-179.960314
C03441=2123.799900,-259.451600,-694.761500,-88.458954,1.936597,-179.948855
C03442=2135.773100,-259.596500,-694.761500,-88.373010,1.959516,-179.943125
C03443=1821.995300,-259.699600,-694.761500,-91.352391,-3.025217,-179.925936
C03444=1827.408200,-259.856700,-694.761500,-90.974239,-2.710090,-179.954584
C03445=2146.457100,-259.907300,-694.761500,-88.275607,2.435071,-179.925936
C03446=1817.310900,-260.023600,-694.761500,-90.922673,-2.589769,-179.960314
C03447=1816.417600,-260.092500,-694.761500,-90.979968,-2.859059,-179.948855
C03448=1829.021700,-260.137100,-694.761500,-91.713354,-2.715820,-179.920207
C03449=1812.424600,-260.433000,-694.761500,-91.661788,-2.738738,-179.920207
C03450=1805.310100,-260.506700,-694.761500,-90.882565,-2.618417,-179.960314
C03451=2155.195100,-260.532700,-694.761500,-89.163692,2.893437,-179.960314
C03452=1801.471000,-260.674000,-694.761500,-91.736273,-2.876248,-179.914477
C03453=2161.924100,-260.829700,-694.761500,-88.768351,1.896490,-179.960314
C03454=2173.333400,-260.918800,-694.761500,-88.791270,3.695578,-179.920207
C03455=1793.567400,-261.027100,-694.761500,-93.352014,18.867500,178.917531
C03456=1798.268100,-261.151000,-694.761500,-91.501360,-2.887707,-179.925936
C03457=2177.388400,-261.248600,-694.761500,-89.576222,3.053865,-179.977503
C03458=2174.096400,-261.393200,-694.761500,-88.968886,3.042406,-179.943125
C03459=1805.813400,-261.482400,-694.761500,-90.773703,-3.707037,-179.948855
C03460=1795.196700,-261.623300,-694.761500,-89.897078,6.554637,-179.988962
C03461=1793.535900,-261.809100,-694.761500,-92.080047,8.548530,179.691024
C03462=2183.607500,-261.944900,-694.761500,-89.266824,3.317426,-179.960314
C03463=2186.836200,-262.175700,-694.761500,-88.676678,3.821628,-179.914477
C03464=2191.049500,-262.383900,-694.761500,-88.705326,-2.400693,179.943125
C03465=2192.205000,-262.721900,-744.761500,-89.272554,-9.230350,179.885829
C03466=2186.150500,-262.552000,-744.761500,-89.576222,2.062648,-179.983232
C03467=2181.639900,-262.451000,-744.761500,-89.163692,2.114214,-179.971773
C03468=2188.040600,-262.361100,-744.761500,-90.464306,2.154321,179.983232
C03469=2193.286900,-262.254400,-744.761500,-90.727867,-16.014170,-179.799886
C03470=2169.038600,-262.158100,-744.761500,-89.175151,1.151645,-179.983232
C03471=2174.293600,-262.023300,-744.761500,-89.186610,1.930868,-179.971773
C03472=2165.569500,-261.801000,-744.761500,-89.129315,1.753251,-179.971773
C03473=2172.003300,-261.704700,-744.761500,-88.762622,2.669983,-179.943125
C03474=2147.913300,-261.463100,-744.761500,-88.556357,1.501149,-179.960314
C03475=2168.241800,-261.324600,-744.761500,-88.785540,2.715820,-179.943125
C03476=2154.272800,-261.123200,-744.761500,-88.882943,1.621471,-179.966043
C03477=1792.665700,-261.053700,-744.761500,-89.255365,1.398017,-179.983232
C03478=2155.862200,-260.871900,-744.761500,-88.642300,2.211617,-179.948855
C03479=1796.126700,-260.757700,-744.761500,-89.604870,-0.945380,179.994691
C03480=2123.757300,-260.664500,-744.761500,-88.596464,1.243318,-179.971773
C03481=2117.710800,-260.542500,-744.761500,-88.779810,2.245995,-179.954584
C03482=1801.190700,-260.462100,-744.761500,-91.392498,-2.824682,-179.931666
C03483=1801.380100,-260.343800,-744.761500,-90.859647,-4.062271,-179.937396
C03484=2101.597900,-260.278300,-744.761500,-88.172475,1.506879,-179.954584
C03485=2132.904900,-260.187400,-744.761500,-87.822971,2.801764,-179.891559
C03486=1813.726800,-260.135700,-744.761500,-88.166746,-3.936220,179.874370
C03487=1808.886200,-260.039800,-744.761500,-91.272177,-2.847600,-179.937396
C03488=2103.586300,-259.955700,-744.761500,-88.395929,1.346451,-179.960314
C03489=2086.875600,-259.846900,-744.761500,-88.659489,0.681820,-179.983232
C03490=2080.363100,-259.763400,-744.761500,-88.625112,1.157375,-179.971773
C03491=2126.908900,-259.735000,-744.761500,-89.089208,1.552716,-179.977503
C03492=2076.632600,-259.653600,-744.761500,-88.143827,1.415206,-179.954584
C03493=2111.703900,-259.551900,-744.761500,-88.533439,1.644389,-179.960314
C03494=1819.587200,-259.478600,-744.761500,-89.919996,-2.320479,179.994691
C03495=2087.002500,-259.406700,-744.761500,-87.880267,1.730333,-179.937396
C03496=1829.709300,-259.351600,-744.761500,-91.953997,-1.839195,-179.937396
C03497=2089.688700,-259.293100,-744.761500,-88.825647,1.392287,-179.971773
C03498=2050.477700,-259.157200,-744.761500,-88.493331,1.019865,-179.971773
C03499=2020.707700,-259.116400,-744.761500,-88.693867,0.664631,-179.983232
C03500=2081.959100,-259.083700,-744.761500,-88.390199,0.721927,-179.977503
C03501=2035.782000,-259.045500,-744.761500,-88.390199,0.962569,-179.971773
C03502=1831.597400,-259.024900,-744.761500,-90.418470,-1.289155,-179.988962
C03503=1829.652500,-258.983000,-744.761500,-90.653382,-2.543933,-179.971773
C03504=2085.385300,-258.913400,-744.761500,-88.659489,1.249048,-179.971773
C03505=1834.984600,-258.872900,-744.761500,-89.627788,-1.558445,179.988962
C03506=2030.140900,-258.831600,-744.761500,-89.106396,0.618794,-179.988962
C03507=1840.317000,-258.770500,-744.761500,-89.381416,-1.357910,179.983232
C03508=2016.519400,-258.730600,-744.761500,-88.264148,0.487014,-179.983232
C03509=2020.124400,-258.703600,-744.761500,-89.220988,0.211994,-179.994691
C03510=2078.781700,-258.633300,-744.761500,-88.504791,0.704738,-179.983232
C03511=1846.044800,-258.566400,-744.761500,-89.341309,-1.014135,179.988962
C03512=2050.036100,-258.547800,-744.761500,-88.602193,1.054242,-179.971773
C03513=2016.344300,-258.493800,-744.761500,-87.817241,0.784952,-179.971773
C03514=2075.622800,-258.456000,-744.761500,-88.585005,1.340721,-179.966043
C03515=1959.820000,-258.437400,-744.761500,-88.585005,0.229183,-179.994691
C03516=1850.469400,-258.397500,-744.761500,-89.828323,-1.449583,179.994691
C03517=1915.896600,-258.375900,-744.761500,-89.135044,0.676090,-179.988962
C03518=1972.664400,-258.348200,-744.761500,-88.808458,1.071431,-179.977503
C03519=2054.245900,-258.323500,-744.761500,-88.865754,0.762034,-179.983232
C03520=2020.202300,-258.300200,-744.761500,-88.476143,0.647442,-179.983232
C03521=2015.024700,-258.274900,-744.761500,-88.436036,0.441178,-179.988962
C03522=2029.853500,-258.244500,-744.761500,-88.636571,0.676090,-179.983232
C03523=2057.358400,-258.226600,-744.761500,-88.882943,0.584417,-179.988962
C03524=1911.051200,-258.195100,-744.761500,-89.255365,0.641713,-179.988962
C03525=1936.591900,-258.183600,-744.761500,-88.860024,-0.005730,180.000421
C03526=1858.586300,-258.172200,-744.761500,-89.690813,-0.744845,179.994691
C03527=1932.976100,-258.144500,-744.761500,-88.579275,0.527121,-179.988962
C03528=1906.246100,-258.108000,-744.761500,-88.871484,0.395341,-179.994691
C03529=1918.700000,-258.096500,-744.761500,-89.243906,-0.108862,180.000421
C03530=1980.001600,-258.069500,-744.761500,-88.670948,0.286479,-179.994691
C03531=1870.966000,-258.056800,-744.761500,-90.401281,-0.630254,-179.994691
C03532=1963.317300,-258.035300,-744.761500,-89.094937,0.320856,-179.994691
C03533=2030.423100,-258.015700,-744.761500,-88.837106,0.693279,-179.983232
C03534=1874.111300,-257.995800,-744.761500,-89.553303,-0.951110,179.994691
C03535=1938.111500,-257.968100,-744.761500,-89.014723,0.223454,-179.994691
C03536=2035.150800,-257.947200,-744.761500,-88.464684,0.527121,-179.983232
C03537=1904.766900,-257.936000,-744.761500,-89.432982,0.429718,-179.994691
C03538=1868.591700,-257.915100,-744.761500,-90.378363,-0.401070,-179.994691
C03539=1875.475100,-257.899500,-744.761500,-89.490278,-0.572958,179.994691
C03540=1879.774100,-257.883000,-744.761500,-89.650706,-0.767763,179.994691
C03541=1945.942000,-257.865700,-744.761500,-89.261095,-0.080214,180.000421
C03542=1906.664000,-257.854900,-744.761500,-88.229771,0.383882,-179.988962
C03543=2006.708400,-257.818400,-744.761500,-88.825647,0.320856,-179.994691
C03544=1880.225100,-257.788000,-744.761500,-90.126261,-0.882355,-180.000421
C03545=1887.098800,-257.749200,-744.761500,-90.046047,-0.446907,-180.000421
C03546=1955.918000,-257.721500,-744.761500,-89.455901,0.309397,-179.994691
C03547=1908.610300,-257.706600,-744.761500,-89.685084,0.876625,-179.994691
C03548=1975.423700,-257.675900,-744.761500,-88.877213,0.664631,-179.988962
C03549=1991.854600,-257.647500,-744.761500,-88.487602,-0.131780,179.994691
C03550=1978.717000,-257.616400,-744.761500,-89.238177,0.796411,-179.988962
C03551=1913.011400,-257.601900,-744.761500,-89.564763,0.063025,-180.000421
C03552=1904.920200,-257.573500,-744.761500,-89.175151,0.481285,-179.994691
C03553=1929.098500,-257.487000,-744.761500,-89.112126,0.607335,-179.988962
C03554=1912.172800,-258.186400,-794.761500,-89.054830,0.750575,-179.988962
C03555=1925.912100,-258.283700,-794.761500,-88.573546,0.853707,-179.977503
C03556=1922.180600,-258.360700,-794.761500,-88.344362,0.017189,-180.000421
C03557=1905.305700,-258.414700,-794.761500,-88.567816,-0.200535,179.994691
C03558=1901.405200,-258.464100,-794.761500,-88.292796,-1.426665,179.960314
C03559=1898.894900,-258.540800,-794.761500,-88.229771,0.315127,-179.988962
C03560=1912.274000,-258.566100,-794.761500,-88.745433,0.572958,-179.988962
C03561=1862.819100,-258.591800,-794.761500,-89.278284,-0.475555,179.994691
C03562=1932.338200,-258.627600,-794.761500,-89.725191,1.100079,-179.994691
C03563=1856.640100,-258.659300,-794.761500,-88.968886,-0.928192,179.983232
C03564=1895.904100,-258.695500,-794.761500,-87.851619,0.269290,-179.988962
C03565=1862.762600,-258.724900,-794.761500,-88.665219,-1.271966,179.971773
C03566=1852.799100,-258.748200,-794.761500,-88.688137,-0.412530,179.988962
C03567=1950.310600,-258.790800,-794.761500,-88.550627,0.160428,-179.994691
C03568=1886.447000,-258.838400,-794.761500,-88.275607,0.338045,-179.988962
C03569=1922.742800,-258.877900,-794.761500,-88.052154,0.699009,-179.977503
C03570=1963.866000,-258.943800,-794.761500,-88.046424,0.429718,-179.983232
C03571=1916.121800,-258.969100,-794.761500,-88.218312,0.338045,-179.988962
C03572=1969.599200,-259.017500,-794.761500,-88.602193,0.309397,-179.994691
C03573=1937.418600,-259.031000,-794.761500,-88.401658,0.727656,-179.977503
C03574=1863.023700,-259.062000,-794.761500,-88.023506,-0.343775,179.988962
C03575=1940.514400,-259.076900,-794.761500,-87.840160,0.234913,-179.988962
C03576=1829.875300,-259.101200,-794.761500,-88.974616,-2.572581,179.954584
C03577=1972.726100,-259.136000,-794.761500,-88.974616,0.693279,-179.988962
C03578=2026.021400,-259.161000,-794.761500,-88.355822,0.796411,-179.977503
C03579=1894.755300,-259.206000,-794.761500,-88.670948,0.624524,-179.983232
C03580=1962.433300,-259.232700,-794.761500,-88.241230,0.217724,-179.994691
C03581=1835.182200,-259.252900,-794.761500,-88.997534,-1.690225,179.971773
C03582=1851.100300,-259.295200,-794.761500,-88.487602,-0.280749,179.994691
C03583=1976.931000,-259.313700,-794.761500,-88.579275,0.974028,-179.977503
C03584=1827.869000,-259.335400,-794.761500,-88.287067,-1.770440,179.948855
C03585=2007.792700,-259.364800,-794.761500,-88.401658,0.183346,-179.994691
C03586=1853.733500,-259.390400,-794.761500,-87.920374,0.229183,-179.988962
C03587=1890.161800,-259.432700,-794.761500,-87.719838,-0.389611,179.983232
C03588=1977.901600,-259.463400,-794.761500,-88.453224,1.140186,-179.971773
C03589=1920.688100,-259.483300,-794.761500,-87.204176,-0.366693,179.983232
C03590=2036.104400,-259.514100,-794.761500,-88.281337,1.071431,-179.966043
C03591=1941.936100,-259.539100,-794.761500,-89.186610,0.641713,-179.988962
C03592=1818.993000,-259.564400,-794.761500,-89.708002,-1.524068,179.994691
C03593=2042.280600,-259.615300,-794.761500,-89.077748,0.796411,-179.988962
C03594=1988.842300,-259.635000,-794.761500,-88.516250,0.830789,-179.977503
C03595=1822.927700,-259.668500,-794.761500,-89.564763,-1.655848,179.988962
C03596=1931.748800,-259.690100,-794.761500,-87.960481,0.487014,-179.983232
C03597=2029.001200,-259.709400,-794.761500,-88.315715,0.555769,-179.983232
C03598=1950.215500,-259.725200,-794.761500,-89.043371,0.206265,-179.994691
C03599=2040.530200,-259.761700,-794.761500,-88.842836,0.515662,-179.988962
C03600=2076.219600,-259.807000,-794.761500,-88.562086,1.197482,-179.971773
C03601=1826.829000,-259.819500,-794.761500,-87.931833,-2.217347,179.920207
C03602=2024.673000,-259.852900,-794.761500,-88.481872,1.037054,-179.971773
C03603=1810.410200,-259.909000,-794.761500,-89.037641,-3.225752,179.943125
C03604=1817.354800,-259.941500,-794.761500,-89.112126,-2.578310,179.960314
C03605=2007.475300,-259.980300,-794.761500,-88.132368,0.315127,-179.988962
C03606=2052.007800,-260.040500,-794.761500,-87.840160,0.922462,-179.966043
C03607=2019.769200,-260.101600,-794.761500,-88.332903,0.658901,-179.983232
C03608=1809.239600,-260.131300,-794.761500,-88.688137,-2.228806,179.948855
C03609=2063.012800,-260.210000,-794.761500,-88.309985,1.501149,-179.954584
C03610=1811.332300,-260.239800,-794.761500,-88.350092,-2.429341,179.931666
C03611=2082.390600,-260.264100,-794.761500,-88.292796,0.939651,-179.971773
C03612=2015.932900,-260.309700,-794.761500,-87.971940,0.401070,-179.983232
C03613=1801.737900,-260.369200,-794.761500,-89.799675,-3.941950,179.988962
C03614=1801.507700,-260.406500,-794.761500,-88.745433,-4.457612,179.903018
C03615=2086.162500,-260.454300,-794.761500,-88.252689,1.243318,-179.960314
C03616=2083.119400,-260.522200,-794.761500,-88.264148,1.031324,-179.966043
C03617=1805.983200,-260.569200,-794.761500,-89.094937,-0.452637,179.994691
C03618=2062.755600,-260.613800,-794.761500,-88.808458,1.157375,-179.977503
C03619=2112.692100,-260.672600,-794.761500,-88.665219,1.283425,-179.971773
C03620=2060.016000,-260.696900,-794.761500,-88.304255,0.481285,-179.983232
C03621=1795.785200,-260.743500,-794.761500,-92.326419,-6.485882,-179.736860
C03622=2066.422300,-260.785700,-794.761500,-88.745433,1.140186,-179.977503
C03623=2104.307400,-260.854000,-794.761500,-88.464684,1.094349,-179.971773
C03624=2090.830900,-260.897600,-794.761500,-88.579275,1.392287,-179.966043
C03625=2081.790500,-260.981500,-794.761500,-89.255365,0.567228,-179.994691
C03626=2087.482800,-261.020900,-794.761500,-88.309985,1.747521,-179.948855
C03627=2093.087800,-261.089500,-794.761500,-88.521979,1.398017,-179.966043
C03628=2081.684700,-261.323900,-794.761500,-88.625112,1.678766,-179.960314
C03629=2093.250200,-261.504000,-794.761500,-88.986075,1.071431,-179.983232
C03630=2117.308900,-261.640800,-794.761500,-88.733974,0.653172,-179.983232
C03631=2118.348900,-261.734700,-794.761500,-88.716785,1.346451,-179.971773
C03632=2130.681900,-261.839100,-794.761500,-89.037641,1.546986,-179.971773
C03633=2136.754200,-262.029700,-794.761500,-88.951698,1.764710,-179.966043
C03634=2129.492000,-262.122600,-794.761500,-88.716785,1.621471,-179.966043
C03635=2141.682300,-262.216200,-794.761500,-88.493331,0.704738,-179.983232
C03636=2134.795400,-262.371900,-794.761500,-88.172475,1.122997,-179.966043
C03637=2154.062000,-262.454000,-794.761500,-88.481872,1.312073,-179.966043
C03638=2141.052200,-262.610100,-794.761500,-89.106396,1.254778,-179.983232
C03639=2178.715600,-262.641900,-794.761500,-89.066289,1.707414,-179.971773
C03640=2175.550100,-262.764200,-794.761500,-88.945968,0.578687,-179.988962
C03641=2185.692700,-262.826500,-794.761500,-89.719461,1.993893,-179.988962
C03642=2155.897800,-262.923300,-794.761500,-89.358498,0.968299,-179.988962
C03643=2181.746600,-262.976800,-794.761500,-89.656436,0.005730,-180.000421
C03644=2192.731400,-263.043900,-794.761500,-90.716408,-16.478266,-179.799886
C03645=2178.029000,-263.116900,-794.761500,-89.072019,1.552716,-179.977503
C03646=2179.286900,-263.227000,-794.761500,-90.126261,1.885031,179.994691
C03647=2190.757100,-263.591000,-844.761500,-87.685461,-3.414828,179.862911
C03648=2185.144900,-263.520900,-844.761500,-87.765675,2.091296,-179.920207
C03649=2182.492100,-263.409100,-844.761500,-89.799675,0.618794,-180.000421
C03650=2186.523800,-263.375000,-844.761500,-89.094937,-2.045459,179.966043
C03651=2177.420100,-263.342900,-844.761500,-88.069343,1.667307,-179.943125
C03652=2187.538000,-263.310100,-844.761500,-90.063236,-2.097026,-180.000421
C03653=2174.586100,-263.258400,-844.761500,-89.507467,-0.040107,180.000421
C03654=2160.540400,-263.204000,-844.761500,-90.533061,0.635983,179.994691
C03655=2170.450600,-263.170900,-844.761500,-90.183557,0.653172,180.000421
C03656=2163.047800,-263.163200,-844.761500,-89.284013,0.653172,-179.994691
C03657=2191.940500,-263.109100,-844.761500,-92.561332,-10.055409,-179.553514
C03658=2152.287500,-263.078400,-844.761500,-89.656436,0.853707,-179.994691
C03659=2155.868500,-263.018200,-844.761500,-89.828323,1.002676,-179.994691
C03660=2155.833600,-262.942500,-844.761500,-88.991805,1.300614,-179.977503
C03661=2143.662400,-262.894900,-844.761500,-89.536115,0.590147,-179.994691
C03662=2130.951000,-262.800000,-844.761500,-89.811134,0.928192,-179.994691
C03663=2127.654800,-262.697300,-844.761500,-89.564763,1.197482,-179.988962
C03664=2124.265200,-262.607100,-844.761500,-89.478819,0.933921,-179.988962
C03665=2137.349200,-262.491900,-844.761500,-89.375686,1.787628,-179.983232
C03666=2106.626700,-262.429400,-844.761500,-89.862701,0.395341,-180.000421
C03667=2128.163100,-262.370200,-844.761500,-89.129315,1.930868,-179.971773
C03668=2095.749300,-262.317200,-844.761500,-89.891348,0.681820,-180.000421
C03669=2064.893600,-262.239200,-844.761500,-78.798886,0.275020,-179.943125
C03670=2076.667800,-262.148600,-844.761500,-82.574677,0.830789,-179.891559
C03671=2099.503100,-262.079000,-844.761500,-88.436036,0.349504,-179.988962
C03672=2066.867400,-261.967900,-844.761500,-90.172098,0.452637,180.000421
C03673=2100.608300,-261.919900,-844.761500,-87.731298,1.535527,-179.937396
C03674=2093.834000,-261.875600,-844.761500,-88.189664,0.962569,-179.971773
C03675=2073.199400,-261.822300,-844.761500,-88.779810,1.025594,-179.977503
C03676=2095.372100,-261.755400,-844.761500,-89.249636,0.985487,-179.988962
C03677=2044.538200,-261.697200,-844.761500,-88.802729,0.475555,-179.988962
C03678=1794.392600,-261.672600,-844.761500,-90.051777,5.987409,179.994691
C03679=2031.188500,-261.603700,-844.761500,-88.155286,0.561499,-179.983232
C03680=2065.564500,-261.557700,-844.761500,-88.785540,0.527121,-179.988962
C03681=1795.779100,-261.522200,-844.761500,-90.195016,3.139809,179.988962
C03682=1807.536300,-261.483700,-844.761500,-77.733184,-1.959516,179.576432
C03683=2015.190600,-261.464100,-844.761500,-86.407765,-0.974028,179.937396
C03684=1832.795400,-261.437100,-844.761500,-79.028069,1.122997,-179.782697
C03685=2040.616300,-261.401600,-844.761500,-88.756892,0.068755,-180.000421
C03686=2004.872100,-261.356000,-844.761500,-88.395929,0.366693,-179.988962
C03687=2027.253800,-261.332700,-844.761500,-89.261095,0.813600,-179.988962
C03688=1817.806900,-261.307000,-844.761500,-89.060560,-1.208941,179.977503
C03689=1979.308900,-261.296900,-844.761500,-88.670948,0.985487,-179.977503
C03690=2005.491100,-261.260800,-844.761500,-88.395929,-0.206265,179.994691
C03691=1903.375800,-261.240800,-844.761500,-83.319523,-0.252101,179.971773
C03692=2053.611200,-261.211800,-844.761500,-88.974616,0.865166,-179.983232
C03693=1805.939400,-261.197400,-844.761500,-89.266824,-1.724603,179.977503
C03694=1840.962800,-261.181000,-844.761500,-83.961235,0.074485,-179.994691
C03695=2021.683200,-261.168200,-844.761500,-88.831377,-0.057296,180.000421
C03696=2041.611100,-261.151300,-844.761500,-88.206853,1.088620,-179.966043
C03697=1978.451500,-261.131000,-844.761500,-88.189664,0.481285,-179.983232
C03698=1959.410800,-261.124300,-844.761500,-88.138098,0.406800,-179.988962
C03699=1915.478400,-261.108000,-844.761500,-88.178205,0.332316,-179.988962
C03700=2018.683200,-261.092800,-844.761500,-88.332903,0.229183,-179.994691
C03701=1817.395600,-261.057700,-844.761500,-88.819917,-0.647442,179.988962
C03702=1934.091100,-261.045200,-844.761500,-88.607923,-0.223454,179.994691
C03703=1964.066300,-261.029300,-844.761500,-88.642300,0.206265,-179.994691
C03704=1996.465000,-261.013100,-844.761500,-88.751162,0.320856,-179.994691
C03705=2036.689300,-260.989100,-844.761500,-88.487602,0.435448,-179.988962
C03706=1895.622100,-260.963800,-844.761500,-87.845889,0.383882,-179.983232
C03707=1866.605300,-260.921600,-844.761500,-88.533439,0.091673,-180.000421
C03708=1823.335500,-260.900600,-844.761500,-89.169422,-0.022918,180.000421
C03709=1897.821400,-260.888800,-844.761500,-87.106774,0.487014,-179.977503
C03710=1814.842100,-260.876300,-844.761500,-88.688137,-0.859437,179.977503
C03711=1908.751800,-260.859100,-844.761500,-88.355822,0.647442,-179.983232
C03712=1917.853000,-260.840800,-844.761500,-87.318768,-0.464096,179.977503
C03713=2051.978200,-260.812800,-844.761500,-88.138098,0.870896,-179.971773
C03714=2013.442000,-260.786800,-844.761500,-87.496385,1.019865,-179.954584
C03715=1842.109500,-260.755300,-844.761500,-88.401658,-0.085944,179.994691
C03716=1974.255200,-260.728600,-844.761500,-87.977669,0.292208,-179.988962
C03717=1810.180700,-260.688400,-844.761500,-90.533061,-1.363640,-179.988962
C03718=1880.062700,-260.642500,-844.761500,-87.794323,-0.005730,180.000421
C03719=1886.132100,-260.630800,-844.761500,-87.960481,-0.532851,179.983232
C03720=1860.965500,-260.620200,-844.761500,-87.742757,-1.334992,179.948855
C03721=1829.201500,-260.590100,-844.761500,-88.986075,-0.968299,179.983232
C03722=2015.480500,-260.569900,-844.761500,-88.716785,0.733386,-179.983232
C03723=1960.755100,-260.516800,-844.761500,-88.224041,0.320856,-179.988962
C03724=2000.074500,-260.492800,-844.761500,-88.659489,-0.349504,179.994691
C03725=1923.633300,-260.478600,-844.761500,-87.926103,0.492744,-179.983232
C03726=1999.131500,-260.425600,-844.761500,-89.129315,-0.091673,180.000421
C03727=1955.933000,-260.396000,-844.761500,-88.436036,1.220400,-179.966043
C03728=1860.273600,-260.365500,-844.761500,-88.132368,-0.269290,179.988962
C03729=1826.611500,-260.346200,-844.761500,-87.668272,-1.678766,179.931666
C03730=1856.873600,-260.288400,-844.761500,-87.920374,0.131780,-179.994691
C03731=1981.193600,-260.241800,-844.761500,-88.367281,0.515662,-179.983232
C03732=1837.269300,-260.199200,-844.761500,-87.639624,-0.446907,179.983232
C03733=1897.160400,-260.176100,-844.761500,-88.923050,-2.102755,179.960314
C03734=1844.001100,-260.130300,-844.761500,-88.510520,-0.830789,179.977503
C03735=1925.927100,-260.081300,-844.761500,-89.100667,-0.131780,180.000421
C03736=1923.028900,-260.032300,-844.761500,-88.877213,0.143239,-179.994691
C03737=1849.043500,-260.005000,-844.761500,-88.464684,-1.117268,179.971773
C03738=1896.208700,-259.952600,-844.761500,-86.447872,-0.177617,179.988962
C03739=1905.085800,-259.917100,-844.761500,-88.487602,0.670361,-179.983232
C03740=1911.597300,-259.838400,-844.761500,-88.854295,-0.452637,179.988962
C03741=1851.855200,-259.744200,-844.761500,-87.943292,-0.762034,179.971773
C03742=1864.571600,-259.658300,-844.761500,-87.874537,-0.378152,179.983232
C03743=2294.292800,-97.327000,-435.033100,7.689094,-78.890559,82.167877
C03744=2292.614600,88.710200,-435.033100,5.145161,-80.231280,84.780565
C03745=2292.553200,217.265700,-435.033100,5.821251,-50.448934,82.471545
C03746=2291.898600,235.641500,-485.033100,80.844345,-89.627788,9.150136
C03747=2292.351100,232.009700,-485.033100,-178.671159,-77.440976,-91.363850
C03748=2291.732900,229.072800,-485.033100,-11.419049,-87.301579,101.430718
C03749=2291.903900,227.580200,-485.033100,-18.076818,-89.438712,108.077029
C03750=2291.747400,224.462500,-485.033100,-0.338045,-89.026182,90.338256
C03751=2291.387700,221.213800,-485.033100,-168.197490,-88.029236,-101.808871
C03752=2291.832400,218.770800,-485.033100,-36.543248,-89.278284,126.543459
C03753=2291.651000,214.508900,-485.033100,162.851794,-84.797754,-72.782829
C03754=2291.701000,212.054100,-485.033100,22.614644,-89.192340,67.385566
C03755=2291.704500,207.896900,-485.033100,41.350364,-89.364227,48.649846
C03756=2291.908400,205.216500,-485.033100,-5.935843,-89.186610,95.936053
C03757=2292.102900,199.366000,-485.033100,131.012529,-89.593410,-41.012319
C03758=2292.040200,196.502400,-485.033100,33.300307,-89.673625,56.699903
C03759=2291.835700,193.347900,-485.033100,-1.254778,-88.407388,91.254988
C03760=2291.654000,187.359300,-485.033100,-172.322786,-86.740081,-97.689304
C03761=2291.982300,182.112500,-485.033100,43.688032,-88.945968,46.306449
C03762=2291.724700,180.272100,-485.033100,174.139063,-86.774458,-84.133123
C03763=2291.862400,175.385000,-485.033100,57.381723,-89.209529,32.612758
C03764=2292.377700,173.436000,-485.033100,84.952452,-89.135044,5.047758
C03765=2292.020300,170.355100,-485.033100,74.123550,-88.980346,15.870931
C03766=2292.054400,167.354400,-485.033100,27.152470,-89.289743,62.847741
C03767=2292.155500,164.346900,-485.033100,23.634509,-89.077748,66.359972
C03768=2291.940800,162.452900,-485.033100,-12.708204,-88.980346,102.708414
C03769=2292.070100,159.090000,-485.033100,40.960753,-88.842836,49.033728
C03770=2292.374200,155.481600,-485.033100,46.581469,-88.951698,43.413012
C03771=2292.643500,150.562100,-485.033100,54.339317,-87.983399,35.649434
C03772=2292.692600,147.878200,-485.033100,66.136518,-88.395929,23.852233
C03773=2292.608700,144.217700,-485.033100,169.509564,-78.334790,-79.291629
C03774=2292.429100,141.205400,-485.033100,24.190278,-88.940239,65.804203
C03775=2292.474800,138.497600,-485.033100,27.467597,-88.384469,62.526884
C03776=2292.148900,135.932700,-485.033100,20.706695,-87.227095,69.270597
C03777=2293.058300,132.652500,-485.033100,55.278968,-87.800053,34.704054
C03778=2292.588900,128.871500,-485.033100,59.679284,-88.751162,30.315197
C03779=2293.262200,126.110500,-485.033100,47.011187,-88.837106,42.983294
C03780=2292.203100,123.960800,-485.033100,-16.323568,-82.345494,106.461288
C03781=2292.290300,120.658900,-485.033100,4.314372,-78.483759,85.594165
C03782=2292.187900,117.357900,-485.033100,145.743274,-88.109450,-55.731605
C03783=2293.096900,114.958500,-485.033100,-3.878924,-86.184312,93.884864
C03784=2292.839000,112.849000,-485.033100,18.901878,-87.421900,71.081144
C03785=2293.042600,108.468200,-485.033100,55.496692,-87.977669,34.486330
C03786=2293.352800,106.749500,-485.033100,33.552408,-88.034965,56.436343
C03787=2293.199900,104.141900,-485.033100,45.962674,-87.674002,44.014618
C03788=2292.557500,100.200400,-485.033100,-146.396446,-88.567816,-123.609915
C03789=2293.249600,98.776700,-485.033100,24.379354,-87.651083,65.603668
C03790=2292.589000,94.404200,-485.033100,12.731122,-82.763754,77.171685
C03791=2293.290700,92.461400,-485.033100,31.186093,-87.049478,58.785470
C03792=2292.827500,88.965700,-485.033100,18.569562,-88.487602,71.424919
C03793=2293.413100,85.313900,-485.033100,9.751742,-88.063613,80.242739
C03794=2293.712500,83.984700,-485.033100,33.157068,-87.937562,56.825954
C03795=2293.144000,79.670200,-485.033100,16.541292,-87.467737,73.441730
C03796=2294.240500,78.079900,-485.033100,40.061209,-88.063613,49.921813
C03797=2293.975600,74.247700,-485.033100,37.408414,-88.436036,52.580337
C03798=2294.433300,72.990100,-485.033100,35.093665,-88.097991,54.895086
C03799=2294.162800,69.373900,-485.033100,23.199061,-88.023506,66.789690
C03800=2293.012900,64.714900,-485.033100,9.029815,-88.625112,80.970396
C03801=2293.313000,62.201200,-485.033100,13.470238,-86.992182,76.512784
C03802=2294.198000,58.420600,-485.033100,32.578380,-86.814565,57.381723
C03803=2294.191700,54.652100,-485.033100,29.919856,-86.871861,60.045977
C03804=2293.922600,52.408000,-485.033100,32.692972,-87.324498,57.278591
C03805=2293.273700,48.844500,-485.033100,55.851926,-88.825647,34.142555
C03806=2294.922300,44.264900,-485.033100,27.834290,-88.224041,62.154462
C03807=2293.651500,42.517200,-485.033100,1.930868,-87.588058,88.069343
C03808=2293.944300,37.531900,-485.033100,24.694481,-86.751540,65.271352
C03809=2293.356600,35.529800,-485.033100,-3.283048,-88.407388,93.283259
C03810=2294.564300,30.629100,-485.033100,0.085944,-87.559410,89.914267
C03811=2294.308800,26.734300,-485.033100,25.107011,-87.536492,64.870282
C03812=2293.745600,24.524000,-485.033100,10.467939,-86.316092,79.509353
C03813=2294.574100,19.335600,-485.033100,22.780802,-87.335957,67.196490
C03814=2294.561900,17.105900,-485.033100,17.263218,-87.473467,72.719803
C03815=2295.099700,13.080200,-485.033100,27.267061,-87.433360,62.704501
C03816=2295.219200,7.993200,-485.033100,45.338150,-87.857348,44.639142
C03817=2295.279500,5.609600,-485.033100,-8.170378,-89.421523,98.170589
C03818=2293.612400,2.704100,-485.033100,17.337703,-87.496385,72.651048
C03819=2294.902400,-1.070500,-485.033100,11.476345,-88.161016,78.518136
C03820=2295.322800,-5.393000,-485.033100,0.131780,-87.032289,89.868430
C03821=2293.951600,-6.944800,-485.033100,5.202457,-88.630841,84.797754
C03822=2294.535000,-10.565600,-485.033100,61.042923,-87.020830,28.922909
C03823=2294.787700,-14.200000,-485.033100,10.553883,-87.903185,79.440598
C03824=2294.436900,-17.470500,-485.033100,9.906440,-86.820295,80.076581
C03825=2294.836900,-21.104900,-485.033100,7.723471,-87.845889,82.271010
C03826=2294.544400,-25.036800,-485.033100,5.036299,-87.651083,84.963911
C03827=2294.009400,-28.997700,-485.033100,15.922497,-87.977669,74.066254
C03828=2295.352400,-32.098100,-485.033100,-20.231140,-87.731298,110.242809
C03829=2294.756400,-34.478200,-485.033100,4.165403,-87.238554,85.829078
C03830=2294.847700,-38.990800,-485.033100,7.333860,-87.467737,82.654892
C03831=2294.463200,-40.495600,-485.033100,-11.321646,-87.599517,101.333316
C03832=2294.755300,-45.282000,-485.033100,4.990462,-87.874537,85.004018
C03833=2295.629100,-49.553900,-485.033100,18.609669,-88.951698,71.384812
C03834=2295.642000,-52.918900,-485.033100,-1.008406,-87.817241,91.008616
C03835=2295.500500,-54.901800,-485.033100,-14.152058,-88.315715,104.157998
C03836=2295.252000,-58.826400,-485.033100,-8.158919,-87.708379,98.164859
C03837=2295.496300,-61.169700,-485.033100,-5.637905,-88.115179,95.638115
C03838=2294.062800,-64.325200,-485.033100,-173.617671,-88.143827,-96.388690
C03839=2294.781800,-67.266500,-485.033100,16.959551,-88.476143,73.034930
C03840=2294.247800,-68.748000,-485.033100,9.144406,-85.817619,80.832886
C03841=2294.210000,-72.025400,-485.033100,18.976362,-87.341686,71.000930
C03842=2294.160700,-75.251000,-485.033100,15.017224,-87.977669,74.971527
C03843=2295.177100,-79.893800,-485.033100,-12.805607,-88.728244,102.805817
C03844=2295.013900,-80.956400,-485.033100,8.496964,-88.716785,81.497517
C03845=2294.942100,-85.634500,-485.033100,10.215837,-88.745433,79.784373
C03846=2294.909400,-88.475100,-485.033100,-12.553505,-88.006317,102.565175
C03847=2295.023000,-90.702500,-485.033100,10.003843,-89.094937,79.996367
C03848=2294.669600,-94.180000,-485.033100,-16.638694,-88.281337,106.644634
C03849=2294.449800,-96.907800,-485.033100,-17.933579,-88.069343,107.939519
C03850=2294.497700,-101.147400,-485.033100,-13.693691,-88.550627,103.699631
C03851=2294.396300,-104.886800,-485.033100,40.926375,-89.461630,49.073835
C03852=2294.523200,-108.512400,-485.033100,148.785680,-89.553303,-58.785470
C03853=2294.602000,-110.438500,-485.033100,7.712012,-89.604870,82.288199
C03854=2294.602000,-116.196600,-485.033100,-11.333105,-89.066289,101.333316
C03855=2294.705800,-120.259700,-485.033100,-36.932859,-89.060560,126.938800
C03856=2294.450700,-124.367200,-485.033100,-36.405738,-89.215258,126.405949
C03857=2294.512700,-127.431100,-485.033100,-39.579924,-89.730920,129.580135
C03858=2294.627100,-131.272100,-485.033100,-45.882460,-88.321444,135.894130
C03859=2294.524200,-134.887400,-485.033100,-43.115074,-89.501737,133.115285
C03860=2294.582800,-137.913800,-485.033100,46.392393,-89.444441,43.602088
C03861=2294.499800,-140.604100,-485.033100,133.298631,-89.392875,-43.298421
C03862=2294.466000,-143.984900,-485.033100,113.548776,-89.897078,-23.548565
C03863=2294.274700,-148.669200,-485.033100,-119.822664,-88.745433,-150.183697
C03864=2294.561200,-150.271900,-485.033100,170.168465,-89.094937,-80.168255
C03865=2293.972500,-151.885100,-535.033100,-62.074248,-86.722892,152.114565
C03866=2294.157900,-149.198900,-535.033100,-90.407010,-88.556357,-179.587891
C03867=2294.219500,-146.456500,-535.033100,-73.338598,-87.421900,163.350267
C03868=2294.446500,-144.131900,-535.033100,-20.093630,-89.524655,110.093840
C03869=2294.413400,-141.779100,-535.033100,-77.200333,-87.903185,167.206273
C03870=2294.465300,-139.475000,-535.033100,-80.237010,-88.338633,170.242950
C03871=2294.671100,-135.342800,-535.033100,-87.565140,-87.811512,177.565350
C03872=2294.650100,-133.979300,-535.033100,-83.525787,-87.141151,173.537457
C03873=2294.813300,-130.913700,-535.033100,-83.863832,-88.034965,173.869773
C03874=2294.781100,-126.993300,-535.033100,-49.211345,-88.711055,139.217285
C03875=2295.204200,-123.792500,-535.033100,-67.368378,-87.662543,157.385777
C03876=2294.917700,-118.707300,-535.033100,-77.177415,-88.258419,167.183355
C03877=2295.345400,-115.741000,-535.033100,-75.126226,-88.596464,165.132166
C03878=2295.439200,-111.658500,-535.033100,-91.403957,-88.149557,-178.596674
C03879=2295.560800,-106.995900,-535.033100,-74.650671,-88.046424,164.656611
C03880=2295.783200,-105.052900,-535.033100,-60.825200,-87.668272,150.848328
C03881=2295.560100,-98.117900,-535.033100,-16.942362,-88.487602,106.948302
C03882=2295.402400,-94.997600,-535.033100,-65.666693,-89.031912,155.666903
C03883=2296.195200,-91.274500,-535.033100,-27.490515,-88.069343,117.502185
C03884=2296.142200,-87.327500,-535.033100,-45.126156,-88.350092,135.137826
C03885=2296.182300,-84.375000,-535.033100,-68.817961,-88.665219,158.823901
C03886=2295.600400,-81.342400,-535.033100,-62.028411,-88.092261,152.040081
C03887=2295.842100,-76.965400,-535.033100,-44.490173,-88.499061,134.496113
C03888=2296.237300,-71.690900,-535.033100,-42.828595,-88.877213,132.828806
C03889=2295.572300,-68.743900,-535.033100,-61.690366,-88.585005,151.696306
C03890=2295.977100,-65.485000,-535.033100,-32.240335,-88.986075,122.246275
C03891=2296.323400,-62.043400,-535.033100,-31.936668,-88.550627,121.948337
C03892=2296.580000,-58.878100,-535.033100,-94.159884,-88.682408,-175.840747
C03893=2296.345000,-55.515500,-535.033100,15.630289,-89.049101,74.369922
C03894=2296.476100,-51.611700,-535.033100,-4.595122,-88.688137,94.595332
C03895=2296.481700,-50.230600,-535.033100,-26.659726,-88.905861,116.659937
C03896=2296.123400,-45.546700,-535.033100,7.964113,-89.341309,82.036097
C03897=2296.406000,-43.797000,-535.033100,-0.286479,-88.103720,90.286689
C03898=2296.149900,-38.927000,-535.033100,-18.649776,-88.980346,108.655716
C03899=2295.966900,-37.167100,-535.033100,15.080249,-88.980346,74.919961
C03900=2296.143200,-33.891700,-535.033100,-0.332316,-88.911591,90.332526
C03901=2296.151200,-30.812600,-535.033100,31.369439,-89.478819,58.630771
C03902=2296.583400,-28.963200,-535.033100,-1.959516,-89.547574,91.959726
C03903=2296.783200,-25.497600,-535.033100,11.825849,-89.243906,78.174362
C03904=2296.509900,-23.035400,-535.033100,-8.136001,-88.441765,98.141941
C03905=2296.727700,-19.082200,-535.033100,28.132228,-88.751162,61.862253
C03906=2296.492500,-16.179800,-535.033100,22.969878,-88.865754,67.024603
C03907=2295.801700,-11.724100,-535.033100,0.784952,-87.708379,89.215258
C03908=2296.034100,-10.406300,-535.033100,-66.039115,-86.791647,156.073703
C03909=2296.170800,-7.139400,-535.033100,12.461832,-88.980346,77.532649
C03910=2295.959200,-3.570400,-535.033100,44.908432,-88.756892,45.086049
C03911=2296.380600,-0.366200,-535.033100,19.852988,-88.602193,70.141493
C03912=2295.635000,1.101000,-535.033100,26.126875,-88.344362,63.867605
C03913=2296.259400,5.028700,-535.033100,50.219751,-87.278661,39.746082
C03914=2296.159300,7.869100,-535.033100,20.202492,-88.819917,69.791989
C03915=2295.517900,11.132800,-535.033100,11.304457,-88.390199,78.690024
C03916=2296.364200,14.523300,-535.033100,35.970290,-88.854295,54.024191
C03917=2296.302500,18.099600,-535.033100,63.329025,-87.221365,26.642537
C03918=2295.561900,20.015700,-535.033100,20.534807,-87.891726,69.448214
C03919=2296.163100,24.633200,-535.033100,72.759910,-89.673625,17.240300
C03920=2295.438500,27.438500,-535.033100,39.820567,-88.390199,50.168185
C03921=2295.912100,29.532300,-535.033100,6.405668,-88.745433,83.594542
C03922=2295.344700,33.916400,-535.033100,17.217382,-88.309985,72.777099
C03923=2295.827700,35.693000,-535.033100,95.873028,-88.046424,-5.872817
C03924=2295.187600,39.320300,-535.033100,17.675748,-88.149557,72.313003
C03925=2295.405400,42.422700,-535.033100,34.371738,-88.550627,55.622743
C03926=2295.713800,44.780600,-535.033100,-17.750232,-87.863078,107.761902
C03927=2295.272200,48.316800,-535.033100,20.970255,-87.834430,69.018496
C03928=2295.565100,50.210300,-535.033100,24.946582,-87.897455,65.036439
C03929=2295.442700,53.203000,-535.033100,31.380898,-87.817241,58.602123
C03930=2295.635700,54.942800,-535.033100,102.794358,-89.037641,-12.794148
C03931=2295.445800,59.103800,-535.033100,19.933202,-88.384469,70.061279
C03932=2295.649700,60.543800,-535.033100,41.596736,-88.980346,48.397745
C03933=2295.546900,64.032000,-535.033100,50.913030,-89.306932,39.081451
C03934=2295.478500,67.704900,-535.033100,53.451233,-87.570869,36.526059
C03935=2294.897900,68.889700,-535.033100,62.544073,-88.877213,27.450408
C03936=2295.424200,73.510900,-535.033100,83.279416,-88.659489,6.720795
C03937=2294.435000,75.611300,-535.033100,62.257594,-88.126638,27.731157
C03938=2295.198300,77.875500,-535.033100,51.697982,-88.103720,38.285040
C03939=2294.414400,80.046500,-535.033100,15.034413,-88.012047,74.960068
C03940=2294.481000,83.948000,-535.033100,45.613170,-87.748486,44.364122
C03941=2294.815600,85.836900,-535.033100,57.255672,-87.376064,32.721620
C03942=2294.897900,88.597400,-535.033100,85.559788,-88.149557,4.434693
C03943=2294.146100,91.052500,-535.033100,36.400009,-87.393252,53.571554
C03944=2294.309600,94.251400,-535.033100,61.908090,-88.562086,28.086391
C03945=2294.361800,98.312200,-535.033100,75.653347,-88.945968,14.346863
C03946=2293.833600,103.190700,-535.033100,46.621576,-87.822971,43.361446
C03947=2294.030600,104.951900,-535.033100,43.269773,-87.404712,46.701790
C03948=2294.208800,109.314800,-535.033100,77.607133,-88.544898,12.393077
C03949=2294.130400,112.734800,-535.033100,82.282469,-87.983399,7.712012
C03950=2293.818100,117.209600,-535.033100,39.539817,-87.696920,50.437475
C03951=2293.809400,120.201900,-535.033100,65.248434,-88.109450,24.734588
C03952=2293.380700,123.319900,-535.033100,54.282022,-88.487602,35.706730
C03953=2293.777000,127.082800,-535.033100,67.345459,-88.006317,22.637562
C03954=2293.458400,129.331200,-535.033100,79.635404,-87.376064,10.353347
C03955=2293.320200,132.979200,-535.033100,63.924901,-87.570869,26.058121
C03956=2293.444800,134.870200,-535.033100,57.060867,-88.430306,32.933614
C03957=2293.054900,139.122300,-535.033100,83.394007,-88.510520,6.606203
C03958=2292.913600,140.884500,-535.033100,52.500123,-87.828700,37.482899
C03959=2292.874600,144.749300,-535.033100,43.246854,-88.264148,46.741897
C03960=2293.391100,147.924900,-535.033100,71.419189,-88.430306,18.575292
C03961=2293.263900,150.040800,-535.033100,55.857655,-88.390199,34.131096
C03962=2293.236400,154.714900,-535.033100,88.991805,-88.373010,1.002676
C03963=2293.153800,158.437600,-535.033100,97.420014,-88.579275,-7.414074
C03964=2292.759200,160.651500,-535.033100,37.746460,-88.269878,52.242292
C03965=2292.929600,165.422600,-535.033100,44.266719,-87.674002,45.710573
C03966=2292.375500,168.559100,-535.033100,29.742239,-88.762622,60.252242
C03967=2292.702400,173.200100,-535.033100,77.991015,-89.014723,12.009195
C03968=2292.657100,176.911000,-535.033100,72.966175,-88.882943,17.028306
C03969=2292.451100,180.212800,-535.033100,59.169352,-88.298526,30.819400
C03970=2292.328000,184.688600,-535.033100,54.350776,-89.089208,35.643704
C03971=2292.574500,188.480900,-535.033100,63.626963,-89.026182,26.367518
C03972=2292.232500,191.004600,-535.033100,39.356471,-88.573546,50.638010
C03973=2292.292800,194.555700,-535.033100,71.172817,-88.779810,18.821664
C03974=2292.309200,197.807500,-535.033100,48.793086,-89.318391,41.207125
C03975=2292.395000,202.453500,-535.033100,36.319795,-89.644977,53.680416
C03976=2292.263200,205.011700,-535.033100,13.475967,-89.748109,76.524243
C03977=2292.319700,208.654700,-535.033100,85.055585,-89.238177,4.944626
C03978=2292.205000,214.890200,-535.033100,45.773598,-89.392875,44.220883
C03979=2292.100800,216.833000,-535.033100,-15.922497,-89.673625,105.922708
C03980=2292.179600,220.664500,-535.033100,15.424024,-89.473089,74.570457
C03981=2292.120000,223.151700,-535.033100,-141.572142,-89.415794,-128.434219
C03982=2292.023800,225.071700,-535.033100,-83.520058,-89.576222,173.520268
C03983=2292.179600,229.159300,-535.033100,128.892586,-89.937185,-38.892375
C03984=2292.170200,229.900800,-535.033100,-133.608028,-89.713732,-136.392603
C03985=2292.189300,235.745600,-535.033100,-166.977090,-89.192340,-103.023541
C03986=2291.981900,239.163600,-585.033100,97.162183,-74.627753,-6.909871
C03987=2292.274900,234.980200,-585.033100,88.447495,-88.183934,1.552716
C03988=2292.307300,233.043400,-585.033100,125.472028,-89.450171,-35.471817
C03989=2292.352400,229.127200,-585.033100,96.044915,-89.559033,-6.044705
C03990=2292.323600,224.898900,-585.033100,-14.679179,-89.564763,104.679389
C03991=2292.336400,221.715800,-585.033100,69.591454,-89.536115,20.408757
C03992=2292.350700,220.271200,-585.033100,86.161393,-88.974616,3.838817
C03993=2292.433000,215.336100,-585.033100,39.287716,-88.006317,50.695306
C03994=2292.362900,213.939000,-585.033100,98.703439,-89.031912,-8.703229
C03995=2292.540300,208.304400,-585.033100,86.367658,-89.318391,3.632552
C03996=2292.529500,205.865100,-585.033100,83.451303,-89.381416,6.548908
C03997=2292.484900,201.883300,-585.033100,29.874019,-89.163692,60.120461
C03998=2292.744900,196.278400,-585.033100,115.508291,-88.848565,-25.508081
C03999=2292.803500,192.981400,-585.033100,102.702685,-89.272554,-12.702474
C04000=2292.733100,188.547800,-585.033100,89.209529,-89.576222,0.790682
C04001=2292.809000,185.602100,-585.033100,98.073186,-89.186610,-8.072975
C04002=2293.033500,183.181500,-585.033100,71.487944,-88.378740,18.506537
C04003=2292.907000,179.364100,-585.033100,83.308063,-88.613653,6.692147
C04004=2293.088600,175.667100,-585.033100,80.494841,-88.814188,9.505370
C04005=2293.207100,169.005800,-585.033100,78.563973,-88.630841,11.430508
C04006=2293.554900,165.530400,-585.033100,104.656471,-86.556734,-14.627613
C04007=2293.566400,161.125200,-585.033100,124.486540,-89.163692,-34.486330
C04008=2293.532600,158.198400,-585.033100,105.372668,-88.831377,-15.366728
C04009=2293.600900,154.591200,-585.033100,37.694893,-87.897455,52.288128
C04010=2293.680800,150.227600,-585.033100,64.434834,-88.321444,25.553918
C04011=2293.594300,145.614700,-585.033100,60.922602,-88.441765,29.071879
C04012=2293.977400,140.963900,-585.033100,136.770755,-88.103720,-46.759086
C04013=2293.942900,138.616200,-585.033100,108.140054,-89.180881,-18.139844
C04014=2293.955900,134.144100,-585.033100,71.407730,-88.298526,18.581021
C04015=2294.115000,130.194400,-585.033100,55.439396,-88.516250,34.555085
C04016=2294.031000,126.078700,-585.033100,48.810275,-87.926103,41.172747
C04017=2294.423200,124.661800,-585.033100,99.814977,-88.854295,-9.814767
C04018=2294.286500,120.922500,-585.033100,97.431473,-88.447495,-7.425533
C04019=2294.412700,117.681900,-585.033100,68.267921,-88.562086,21.726560
C04020=2294.499800,112.632500,-585.033100,91.994104,-88.344362,-1.993893
C04021=2294.636100,110.144900,-585.033100,47.555497,-89.295472,42.444713
C04022=2294.647300,105.281900,-585.033100,59.112056,-88.332903,30.876696
C04023=2294.900300,100.337600,-585.033100,78.970773,-88.842836,11.023708
C04024=2294.881100,97.854100,-585.033100,91.971185,-88.659489,-1.970975
C04025=2294.919100,94.649600,-585.033100,123.346354,-88.481872,-33.340414
C04026=2295.117100,92.707300,-585.033100,117.215706,-89.008993,-27.209766
C04027=2295.078400,88.532200,-585.033100,40.720110,-88.521979,49.268641
C04028=2295.239100,85.873400,-585.033100,72.330192,-88.539168,17.664289
C04029=2295.311200,83.452000,-585.033100,67.620479,-88.413117,22.368272
C04030=2295.347500,80.167800,-585.033100,130.645836,-88.395929,-40.634167
C04031=2295.239800,77.128500,-585.033100,79.526542,-88.825647,10.473668
C04032=2295.550400,72.880600,-585.033100,78.581162,-88.241230,11.413319
C04033=2295.641300,69.934600,-585.033100,121.083171,-88.625112,-31.077231
C04034=2295.436000,67.226700,-585.033100,112.735176,-87.742757,-22.723506
C04035=2295.643400,64.450200,-585.033100,149.519066,-88.269878,-59.507397
C04036=2295.652800,61.081000,-585.033100,31.329332,-88.447495,58.659419
C04037=2295.738600,58.576600,-585.033100,143.715004,-89.157963,-53.709064
C04038=2295.778800,53.833500,-585.033100,100.903597,-88.327174,-10.897657
C04039=2295.902700,52.243400,-585.033100,111.537694,-88.539168,-21.531754
C04040=2295.986000,49.210600,-585.033100,111.251215,-88.327174,-21.239545
C04041=2296.018400,45.944600,-585.033100,56.029543,-88.390199,33.959209
C04042=2296.181000,43.243200,-585.033100,122.515565,-89.478819,-32.515355
C04043=2296.085100,39.045400,-585.033100,96.279828,-87.845889,-6.273888
C04044=2296.289300,36.019600,-585.033100,114.356646,-89.639247,-24.356436
C04045=2296.237000,33.376800,-585.033100,110.649609,-88.951698,-20.649399
C04046=2296.293800,29.892300,-585.033100,47.486742,-89.117855,42.507739
C04047=2296.439800,26.554500,-585.033100,127.477380,-88.544898,-37.465710
C04048=2296.365600,23.455800,-585.033100,123.248951,-89.851241,-33.248741
C04049=2296.566700,20.399100,-585.033100,73.017741,-88.550627,16.976739
C04050=2296.334900,18.322500,-585.033100,-158.967140,-89.954374,-111.033491
C04051=2296.461100,15.755700,-585.033100,34.916048,-89.295472,55.084162
C04052=2296.595600,13.590800,-585.033100,119.879959,-89.919996,-29.879749
C04053=2296.455900,10.058000,-585.033100,136.959831,-88.585005,-46.953891
C04054=2296.488300,7.358400,-585.033100,54.035650,-88.882943,35.958831
C04055=2296.602300,3.702800,-585.033100,113.606072,-89.243906,-23.605861
C04056=2296.473600,0.692200,-585.033100,175.399570,-89.736650,-85.399359
C04057=2296.522100,-4.279200,-585.033100,32.372115,-89.157963,57.622365
C04058=2296.634700,-5.925500,-585.033100,55.301886,-89.518926,34.692594
C04059=2296.769600,-11.815800,-585.033100,76.690401,-88.722515,13.309810
C04060=2296.731900,-13.109800,-585.033100,9.138677,-89.564763,80.861534
C04061=2296.716900,-17.512300,-585.033100,14.037466,-89.530385,75.962744
C04062=2296.689100,-19.925200,-585.033100,36.491682,-88.487602,53.497069
C04063=2296.748300,-24.255300,-585.033100,115.731745,-89.289743,-25.731535
C04064=2296.822500,-27.631400,-585.033100,28.126498,-89.467360,61.873712
C04065=2296.834700,-31.536600,-585.033100,-173.915609,-88.825647,-96.085022
C04066=2296.762200,-34.123800,-585.033100,113.376889,-89.599140,-23.376678
C04067=2296.832100,-36.609200,-585.033100,170.466403,-89.690813,-80.466193
C04068=2296.749700,-42.605400,-585.033100,157.127946,-89.438712,-67.127735
C04069=2296.718000,-45.444700,-585.033100,-62.899307,-89.398605,152.905247
C04070=2296.808600,-49.040100,-585.033100,21.686453,-89.387146,68.313758
C04071=2296.862300,-52.064400,-585.033100,-114.809283,-89.834053,-155.191348
C04072=2296.729100,-56.165900,-585.033100,-107.830657,-88.923050,-162.175704
C04073=2296.833700,-59.633600,-585.033100,-24.459568,-89.008993,114.465508
C04074=2296.698500,-63.805300,-585.033100,-119.610669,-88.487602,-150.395692
C04075=2296.716900,-66.061100,-585.033100,-96.142318,-89.387146,-173.858313
C04076=2296.776500,-70.804400,-585.033100,-87.192717,-89.232447,177.192928
C04077=2296.618600,-74.757600,-585.033100,-151.266587,-89.404334,-118.734044
C04078=2296.584800,-78.209300,-585.033100,-111.795525,-89.117855,-158.205106
C04079=2296.415800,-81.194500,-585.033100,-68.852338,-89.536115,158.852549
C04080=2296.491400,-85.241300,-585.033100,-67.637668,-89.524655,157.637878
C04081=2296.306300,-87.454800,-585.033100,-45.876731,-87.914644,135.894130
C04082=2296.346300,-90.589900,-585.033100,-85.817619,-88.355822,175.823559
C04083=2296.145000,-94.229700,-585.033100,-80.443274,-88.458954,170.449214
C04084=2296.228300,-97.578700,-585.033100,-90.160639,-88.034965,-179.839993
C04085=2295.977300,-101.108100,-585.033100,-103.928814,-88.012047,-166.077546
C04086=2295.829500,-105.521800,-585.033100,-78.541055,-87.702650,168.552724
C04087=2295.696000,-110.186500,-585.033100,-60.664771,-88.218312,150.676441
C04088=2295.689100,-112.617300,-585.033100,-100.233237,-86.992182,-169.784583
C04089=2295.489000,-114.766300,-585.033100,-86.253066,-87.754216,176.253277
C04090=2295.378000,-116.803700,-585.033100,-118.522050,-87.616706,-151.495771
C04091=2295.238100,-120.644500,-585.033100,-88.092261,-87.708379,178.092471
C04092=2295.200100,-123.925300,-585.033100,-80.391708,-87.674002,170.397648
C04093=2295.100100,-127.527500,-585.033100,-102.089620,-87.851619,-167.916741
C04094=2295.040800,-130.121200,-585.033100,-95.162560,-87.507844,-174.843801
C04095=2294.840400,-132.883300,-585.033100,-110.850145,-87.610976,-159.167675
C04096=2294.748000,-136.578000,-585.033100,-95.156831,-87.593788,-174.843801
C04097=2294.526700,-139.599700,-585.033100,-89.547574,-87.897455,179.547784
C04098=2294.447900,-143.016300,-585.033100,-103.487637,-87.565140,-166.524454
C04099=2294.440900,-146.593100,-585.033100,-94.136966,-84.631596,-175.880854
C04100=2294.048100,-149.378100,-585.033100,-114.345187,-87.381793,-155.678363
C04101=2293.899800,-150.227300,-585.033100,-94.314583,-88.172475,-175.686049
C04102=2293.062400,-157.986600,-635.033100,-96.933000,-75.819505,-173.273896
C04103=2293.736500,-150.954000,-635.033100,-76.421111,-87.914644,166.432780
C04104=2293.528400,-149.433000,-635.033100,-93.552549,-86.860402,-176.453812
C04105=2294.048700,-146.128200,-635.033100,-100.244696,-86.310362,-169.773124
C04106=2294.120300,-141.917600,-635.033100,-95.454769,-87.175529,-174.551592
C04107=2294.193500,-140.690600,-635.033100,-104.581986,-87.072396,-165.435834
C04108=2294.587700,-137.155000,-635.033100,-158.909844,-87.593788,-111.107976
C04109=2294.266000,-135.971600,-635.033100,-110.403238,-87.450548,-159.614583
C04110=2294.600600,-131.190200,-635.033100,-116.591182,-87.588058,-153.426638
C04111=2294.473700,-128.485200,-635.033100,-113.027384,-86.573923,-157.007625
C04112=2295.015700,-123.870600,-635.033100,-84.115934,-87.983399,174.121874
C04113=2294.814600,-121.629700,-635.033100,-108.289023,-87.129692,-161.734526
C04114=2295.263800,-118.009600,-635.033100,-97.185101,-87.622436,-172.821260
C04115=2295.259700,-115.970600,-635.033100,-106.077406,-87.834430,-163.934684
C04116=2295.283000,-111.760500,-635.033100,-72.261437,-88.894402,162.267377
